gfCNCPoint2[6043] = {X 559.9503, Y 48.1273, Z -2.1667, A 0.000, B 0.000, C 0.000 }
gfCNCPoint2[6044] = {X 559.3170, Y 47.4940, Z -2.1667, A 0.000, B 0.000, C 0.000 }
gfCNCPoint2[6045] = {X 558.8404, Y 46.7355, Z -2.1667, A 0.000, B 0.000, C 0.000 }
gfCNCPoint2[6046] = {X 558.5446, Y 45.8901, Z -2.1667, A 0.000, B 0.000, C 0.000 }
gfCNCPoint2[6047] = {X 558.4443, Y 45.0000, Z -2.1667, A 0.000, B 0.000, C 0.000 }
gfCNCPoint2[6048] = {X 558.4443, Y 44.0660, Z -2.1667, A 0.000, B 0.000, C 0.000 }
gfCNCPoint2[6049] = {X 558.5395, Y 43.2139, Z -2.1667, A 0.000, B 0.000, C 0.000 }
gfCNCPoint2[6050] = {X 558.8124, Y 42.4011, Z -2.1667, A 0.000, B 0.000, C 0.000 }
gfCNCPoint2[6051] = {X 559.2508, Y 41.6643, Z -2.1667, A 0.000, B 0.000, C 0.000 }
gfCNCPoint2[6052] = {X 559.8349, Y 41.0367, Z -2.1667, A 0.000, B 0.000, C 0.000 }
gfCNCPoint2[6053] = {X 559.9032, Y 40.9788, Z -2.1667, A 0.000, B 0.000, C 0.000 }
gfCNCPoint2[6054] = {X 559.9727, Y 40.9224, Z -2.1667, A 0.000, B 0.000, C 0.000 }
gfCNCPoint2[6055] = {X 559.9727, Y 9.0791, Z -2.1667, A 0.000, B 0.000, C 0.000 }
gfCNCPoint2[6056] = {X 559.9026, Y 9.0227, Z -2.1667, A 0.000, B 0.000, C 0.000 }
gfCNCPoint2[6057] = {X 559.8337, Y 8.9647, Z -2.1667, A 0.000, B 0.000, C 0.000 }
gfCNCPoint2[6058] = {X 559.2474, Y 8.3382, Z -2.1667, A 0.000, B 0.000, C 0.000 }
gfCNCPoint2[6059] = {X 558.8082, Y 7.6010, Z -2.1667, A 0.000, B 0.000, C 0.000 }
gfCNCPoint2[6060] = {X 558.5363, Y 6.7871, Z -2.1667, A 0.000, B 0.000, C 0.000 }
gfCNCPoint2[6061] = {X 558.4443, Y 5.9339, Z -2.1667, A 0.000, B 0.000, C 0.000 }
gfCNCPoint2[6062] = {X 558.4443, Y 5.0000, Z -2.1667, A 0.000, B 0.000, C 0.000 }
gfCNCPoint2[6063] = {X 558.5446, Y 4.1099, Z -2.1667, A 0.000, B 0.000, C 0.000 }
gfCNCPoint2[6064] = {X 558.8404, Y 3.2645, Z -2.1667, A 0.000, B 0.000, C 0.000 }
gfCNCPoint2[6065] = {X 559.3170, Y 2.5060, Z -2.1667, A 0.000, B 0.000, C 0.000 }
gfCNCPoint2[6066] = {X 559.9503, Y 1.8727, Z -2.1667, A 0.000, B 0.000, C 0.000 }
gfCNCPoint2[6067] = {X 560.7088, Y 1.3961, Z -2.1667, A 0.000, B 0.000, C 0.000 }
gfCNCPoint2[6068] = {X 561.5542, Y 1.1003, Z -2.1667, A 0.000, B 0.000, C 0.000 }
gfCNCPoint2[6069] = {X 562.4443, Y 1.0000, Z -2.1667, A 0.000, B 0.000, C 0.000 }
gfCNCPoint2[6070] = {X 570.9376, Y 1.0000, Z -2.1667, A 0.000, B 0.000, C 0.000 }
gfCNCPoint2[6071] = {X 571.8276, Y 1.1003, Z -2.1667, A 0.000, B 0.000, C 0.000 }
gfCNCPoint2[6072] = {X 572.6731, Y 1.3961, Z -2.1667, A 0.000, B 0.000, C 0.000 }
gfCNCPoint2[6073] = {X 573.4315, Y 1.8727, Z -2.1667, A 0.000, B 0.000, C 0.000 }
gfCNCPoint2[6074] = {X 574.0649, Y 2.5060, Z -2.1667, A 0.000, B 0.000, C 0.000 }
gfCNCPoint2[6075] = {X 574.5414, Y 3.2645, Z -2.1667, A 0.000, B 0.000, C 0.000 }
gfCNCPoint2[6076] = {X 574.8373, Y 4.1099, Z -2.1667, A 0.000, B 0.000, C 0.000 }
gfCNCPoint2[6077] = {X 574.9376, Y 5.0000, Z -2.1667, A 0.000, B 0.000, C 0.000 }
gfCNCPoint2[6078] = {X 574.9372, Y 5.9858, Z -2.1667, A 0.000, B 0.000, C 0.000 }
gfCNCPoint2[6079] = {X 574.8649, Y 6.6932, Z -2.1667, A 0.000, B 0.000, C 0.000 }
gfCNCPoint2[6080] = {X 574.6684, Y 7.3766, Z -2.1667, A 0.000, B 0.000, C 0.000 }
gfCNCPoint2[6081] = {X 574.3540, Y 8.0145, Z -2.1667, A 0.000, B 0.000, C 0.000 }
gfCNCPoint2[6082] = {X 574.2916, Y 8.1136, Z -2.1667, A 0.000, B 0.000, C 0.000 }
gfCNCPoint2[6083] = {X 574.2264, Y 8.2108, Z -2.1667, A 0.000, B 0.000, C 0.000 }
gfCNCPoint2[6084] = {X 574.2604, Y 8.2360, Z -2.1667, A 0.000, B 0.000, C 0.000 }
gfCNCPoint2[6085] = {X 574.2832, Y 8.2715, Z -2.1667, A 0.000, B 0.000, C 0.000 }
gfCNCPoint2[6086] = {X 574.9161, Y 9.8088, Z -2.1667, A 0.000, B 0.000, C 0.000 }
gfCNCPoint2[6087] = {X 581.1904, Y 25.2176, Z -2.1667, A 0.000, B 0.000, C 0.000 }
gfCNCPoint2[6088] = {X 588.2030, Y 8.0669, Z -2.1667, A 0.000, B 0.000, C 0.000 }
gfCNCPoint2[6089] = {X 587.8648, Y 7.3988, Z -2.1667, A 0.000, B 0.000, C 0.000 }
gfCNCPoint2[6090] = {X 587.6570, Y 6.6794, Z -2.1667, A 0.000, B 0.000, C 0.000 }
gfCNCPoint2[6091] = {X 587.5870, Y 5.9339, Z -2.1667, A 0.000, B 0.000, C 0.000 }
gfCNCPoint2[6092] = {X 587.5870, Y 5.0000, Z -2.1667, A 0.000, B 0.000, C 0.000 }
gfCNCPoint2[6093] = {X 587.6872, Y 4.1099, Z -2.1667, A 0.000, B 0.000, C 0.000 }
gfCNCPoint2[6094] = {X 587.9831, Y 3.2645, Z -2.1667, A 0.000, B 0.000, C 0.000 }
gfCNCPoint2[6095] = {X 588.4596, Y 2.5060, Z -2.1667, A 0.000, B 0.000, C 0.000 }
gfCNCPoint2[6096] = {X 589.0930, Y 1.8727, Z -2.1667, A 0.000, B 0.000, C 0.000 }
gfCNCPoint2[6097] = {X 589.8514, Y 1.3961, Z -2.1667, A 0.000, B 0.000, C 0.000 }
gfCNCPoint2[6098] = {X 590.6969, Y 1.1003, Z -2.1667, A 0.000, B 0.000, C 0.000 }
gfCNCPoint2[6099] = {X 591.5870, Y 1.0000, Z -2.1667, A 0.000, B 0.000, C 0.000 }
gfCNCPoint2[6100] = {X 600.0000, Y 1.0000, Z -2.1667, A 0.000, B 0.000, C 0.000 }
gfCNCPoint2[6101] = {X 600.7927, Y 1.0793, Z -2.1667, A 0.000, B 0.000, C 0.000 }
gfCNCPoint2[6102] = {X 601.5540, Y 1.3142, Z -2.1667, A 0.000, B 0.000, C 0.000 }
gfCNCPoint2[6103] = {X 602.2536, Y 1.6953, Z -2.1667, A 0.000, B 0.000, C 0.000 }
gfCNCPoint2[6104] = {X 602.8638, Y 2.2074, Z -2.1667, A 0.000, B 0.000, C 0.000 }
gfCNCPoint2[6105] = {X 603.3604, Y 2.8303, Z -2.1667, A 0.000, B 0.000, C 0.000 }
gfCNCPoint2[6106] = {X 603.5430, Y 3.1434, Z -2.1667, A 0.000, B 0.000, C 0.000 }
gfCNCPoint2[6107] = {X 603.6965, Y 3.4716, Z -2.1667, A 0.000, B 0.000, C 0.000 }
gfCNCPoint2[6108] = {X 607.6965, Y 13.1458, Z -2.1667, A 0.000, B 0.000, C 0.000 }
gfCNCPoint2[6109] = {X 607.6965, Y 13.1458, Z 0.8333, A 0.000, B 0.000, C 0.000 }
gfCNCPoint2[6110] = {X 607.6965, Y 13.1458, Z 11.0000, A 0.000, B 0.000, C 0.000 }
gfCNCPoint2[6111] = {X 448.7118, Y 19.7811, Z 11.0000, A 0.000, B 0.000, C 0.000 }
gfCNCPoint2[6112] = {X 448.7118, Y 19.7811, Z 1.6667, A 0.000, B 0.000, C 0.000 }
gfCNCPoint2[6113] = {X 444.0413, Y 19.7808, Z 0.4152, A 0.000, B 0.000, C 0.000 }
gfCNCPoint2[6114] = {X 443.3489, Y 19.7970, Z 0.2296, A 0.000, B 0.000, C 0.000 }
gfCNCPoint2[6115] = {X 442.7481, Y 19.8041, Z 0.0686, A 0.000, B 0.000, C 0.000 }
gfCNCPoint2[6116] = {X 442.0371, Y 19.9272, Z -0.1247, A 0.000, B 0.000, C 0.000 }
gfCNCPoint2[6117] = {X 441.4689, Y 20.1225, Z -0.2857, A 0.000, B 0.000, C 0.000 }
gfCNCPoint2[6118] = {X 441.3658, Y 20.1579, Z -0.3149, A 0.000, B 0.000, C 0.000 }
gfCNCPoint2[6119] = {X 441.3328, Y 20.2618, Z -0.3441, A 0.000, B 0.000, C 0.000 }
gfCNCPoint2[6120] = {X 441.1879, Y 20.7173, Z -0.4722, A 0.000, B 0.000, C 0.000 }
gfCNCPoint2[6121] = {X 441.1541, Y 21.8891, Z -0.7863, A 0.000, B 0.000, C 0.000 }
gfCNCPoint2[6122] = {X 441.2726, Y 22.3522, Z -0.9144, A 0.000, B 0.000, C 0.000 }
gfCNCPoint2[6123] = {X 441.5010, Y 22.4270, Z -0.9788, A 0.000, B 0.000, C 0.000 }
gfCNCPoint2[6124] = {X 441.7404, Y 22.4490, Z -1.0432, A 0.000, B 0.000, C 0.000 }
gfCNCPoint2[6125] = {X 442.9814, Y 22.5631, Z -1.3771, A 0.000, B 0.000, C 0.000 }
gfCNCPoint2[6126] = {X 443.1437, Y 22.5696, Z -1.4207, A 0.000, B 0.000, C 0.000 }
gfCNCPoint2[6127] = {X 444.3942, Y 22.5560, Z -1.7558, A 0.000, B 0.000, C 0.000 }
gfCNCPoint2[6128] = {X 445.9278, Y 22.5560, Z -2.1667, A 0.000, B 0.000, C 0.000 }
gfCNCPoint2[6129] = {X 450.1184, Y 22.5560, Z -2.1667, A 0.000, B 0.000, C 0.000 }
gfCNCPoint2[6130] = {X 450.1184, Y 19.7812, Z -2.1667, A 0.000, B 0.000, C 0.000 }
gfCNCPoint2[6131] = {X 444.0413, Y 19.7808, Z -2.1667, A 0.000, B 0.000, C 0.000 }
gfCNCPoint2[6132] = {X 443.3489, Y 19.7970, Z -2.1667, A 0.000, B 0.000, C 0.000 }
gfCNCPoint2[6133] = {X 442.3959, Y 19.8846, Z -2.1667, A 0.000, B 0.000, C 0.000 }
gfCNCPoint2[6134] = {X 441.4689, Y 20.1225, Z -2.1667, A 0.000, B 0.000, C 0.000 }
gfCNCPoint2[6135] = {X 441.3843, Y 20.1760, Z -2.1667, A 0.000, B 0.000, C 0.000 }
gfCNCPoint2[6136] = {X 441.3328, Y 20.2618, Z -2.1667, A 0.000, B 0.000, C 0.000 }
gfCNCPoint2[6137] = {X 441.1824, Y 20.9508, Z -2.1667, A 0.000, B 0.000, C 0.000 }
gfCNCPoint2[6138] = {X 441.1621, Y 21.6557, Z -2.1667, A 0.000, B 0.000, C 0.000 }
gfCNCPoint2[6139] = {X 441.2726, Y 22.3522, Z -2.1667, A 0.000, B 0.000, C 0.000 }
gfCNCPoint2[6140] = {X 441.5038, Y 22.4137, Z -2.1667, A 0.000, B 0.000, C 0.000 }
gfCNCPoint2[6141] = {X 441.7404, Y 22.4490, Z -2.1667, A 0.000, B 0.000, C 0.000 }
gfCNCPoint2[6142] = {X 443.0660, Y 22.5366, Z -2.1667, A 0.000, B 0.000, C 0.000 }
gfCNCPoint2[6143] = {X 444.3942, Y 22.5560, Z -2.1667, A 0.000, B 0.000, C 0.000 }
gfCNCPoint2[6144] = {X 445.9278, Y 22.5560, Z -2.1667, A 0.000, B 0.000, C 0.000 }
gfCNCPoint2[6145] = {X 441.9430, Y 22.2874, Z -2.1667, A 0.000, B 0.000, C 0.000 }
gfCNCPoint2[6146] = {X 445.9278, Y 22.6360, Z -2.1667, A 0.000, B 0.000, C 0.000 }
gfCNCPoint2[6147] = {X 450.1984, Y 22.6360, Z -2.1667, A 0.000, B 0.000, C 0.000 }
gfCNCPoint2[6148] = {X 450.1984, Y 19.7012, Z -2.1667, A 0.000, B 0.000, C 0.000 }
gfCNCPoint2[6149] = {X 444.0404, Y 19.7008, Z -2.1667, A 0.000, B 0.000, C 0.000 }
gfCNCPoint2[6150] = {X 443.3498, Y 19.7169, Z -2.1667, A 0.000, B 0.000, C 0.000 }
gfCNCPoint2[6151] = {X 442.3831, Y 19.8056, Z -2.1667, A 0.000, B 0.000, C 0.000 }
gfCNCPoint2[6152] = {X 441.4429, Y 20.0469, Z -2.1667, A 0.000, B 0.000, C 0.000 }
gfCNCPoint2[6153] = {X 441.3271, Y 20.1201, Z -2.1667, A 0.000, B 0.000, C 0.000 }
gfCNCPoint2[6154] = {X 441.2566, Y 20.2375, Z -2.1667, A 0.000, B 0.000, C 0.000 }
gfCNCPoint2[6155] = {X 441.1012, Y 20.9555, Z -2.1667, A 0.000, B 0.000, C 0.000 }
gfCNCPoint2[6156] = {X 441.0842, Y 21.6898, Z -2.1667, A 0.000, B 0.000, C 0.000 }
gfCNCPoint2[6157] = {X 441.2061, Y 22.4142, Z -2.1667, A 0.000, B 0.000, C 0.000 }
gfCNCPoint2[6158] = {X 441.4661, Y 22.4875, Z -2.1667, A 0.000, B 0.000, C 0.000 }
gfCNCPoint2[6159] = {X 441.7331, Y 22.5286, Z -2.1667, A 0.000, B 0.000, C 0.000 }
gfCNCPoint2[6160] = {X 443.0614, Y 22.6165, Z -2.1667, A 0.000, B 0.000, C 0.000 }
gfCNCPoint2[6161] = {X 444.3925, Y 22.6360, Z -2.1667, A 0.000, B 0.000, C 0.000 }
gfCNCPoint2[6162] = {X 445.9278, Y 22.6360, Z -2.1667, A 0.000, B 0.000, C 0.000 }
gfCNCPoint2[6163] = {X 449.9125, Y 22.2874, Z -2.1667, A 0.000, B 0.000, C 0.000 }
gfCNCPoint2[6164] = {X 441.9430, Y 22.3674, Z -2.1667, A 0.000, B 0.000, C 0.000 }
gfCNCPoint2[6165] = {X 445.9278, Y 22.7160, Z -2.1667, A 0.000, B 0.000, C 0.000 }
gfCNCPoint2[6166] = {X 450.2784, Y 22.7160, Z -2.1667, A 0.000, B 0.000, C 0.000 }
gfCNCPoint2[6167] = {X 450.2784, Y 19.6212, Z -2.1667, A 0.000, B 0.000, C 0.000 }
gfCNCPoint2[6168] = {X 444.0395, Y 19.6208, Z -2.1667, A 0.000, B 0.000, C 0.000 }
gfCNCPoint2[6169] = {X 443.3484, Y 19.6370, Z -2.1667, A 0.000, B 0.000, C 0.000 }
gfCNCPoint2[6170] = {X 442.3693, Y 19.7268, Z -2.1667, A 0.000, B 0.000, C 0.000 }
gfCNCPoint2[6171] = {X 441.4169, Y 19.9712, Z -2.1667, A 0.000, B 0.000, C 0.000 }
gfCNCPoint2[6172] = {X 441.2699, Y 20.0642, Z -2.1667, A 0.000, B 0.000, C 0.000 }
gfCNCPoint2[6173] = {X 441.1803, Y 20.2133, Z -2.1667, A 0.000, B 0.000, C 0.000 }
gfCNCPoint2[6174] = {X 441.0202, Y 20.9599, Z -2.1667, A 0.000, B 0.000, C 0.000 }
gfCNCPoint2[6175] = {X 441.0065, Y 21.7235, Z -2.1667, A 0.000, B 0.000, C 0.000 }
gfCNCPoint2[6176] = {X 441.1399, Y 22.4754, Z -2.1667, A 0.000, B 0.000, C 0.000 }
gfCNCPoint2[6177] = {X 441.4285, Y 22.5611, Z -2.1667, A 0.000, B 0.000, C 0.000 }
gfCNCPoint2[6178] = {X 441.7258, Y 22.6083, Z -2.1667, A 0.000, B 0.000, C 0.000 }
gfCNCPoint2[6179] = {X 443.0580, Y 22.6964, Z -2.1667, A 0.000, B 0.000, C 0.000 }
gfCNCPoint2[6180] = {X 444.3929, Y 22.7160, Z -2.1667, A 0.000, B 0.000, C 0.000 }
gfCNCPoint2[6181] = {X 445.9278, Y 22.7160, Z -2.1667, A 0.000, B 0.000, C 0.000 }
gfCNCPoint2[6182] = {X 449.9125, Y 22.3674, Z -2.1667, A 0.000, B 0.000, C 0.000 }
gfCNCPoint2[6183] = {X 441.9430, Y 22.4474, Z -2.1667, A 0.000, B 0.000, C 0.000 }
gfCNCPoint2[6184] = {X 445.9278, Y 22.7960, Z -2.1667, A 0.000, B 0.000, C 0.000 }
gfCNCPoint2[6185] = {X 450.3584, Y 22.7960, Z -2.1667, A 0.000, B 0.000, C 0.000 }
gfCNCPoint2[6186] = {X 450.3584, Y 19.5412, Z -2.1667, A 0.000, B 0.000, C 0.000 }
gfCNCPoint2[6187] = {X 444.0385, Y 19.5408, Z -2.1667, A 0.000, B 0.000, C 0.000 }
gfCNCPoint2[6188] = {X 443.3470, Y 19.5570, Z -2.1667, A 0.000, B 0.000, C 0.000 }
gfCNCPoint2[6189] = {X 442.3554, Y 19.6480, Z -2.1667, A 0.000, B 0.000, C 0.000 }
gfCNCPoint2[6190] = {X 441.3909, Y 19.8955, Z -2.1667, A 0.000, B 0.000, C 0.000 }
gfCNCPoint2[6191] = {X 441.2127, Y 20.0083, Z -2.1667, A 0.000, B 0.000, C 0.000 }
gfCNCPoint2[6192] = {X 441.1041, Y 20.1890, Z -2.1667, A 0.000, B 0.000, C 0.000 }
gfCNCPoint2[6193] = {X 440.9392, Y 20.9642, Z -2.1667, A 0.000, B 0.000, C 0.000 }
gfCNCPoint2[6194] = {X 440.9290, Y 21.7567, Z -2.1667, A 0.000, B 0.000, C 0.000 }
gfCNCPoint2[6195] = {X 441.0740, Y 22.5359, Z -2.1667, A 0.000, B 0.000, C 0.000 }
gfCNCPoint2[6196] = {X 441.3909, Y 22.6345, Z -2.1667, A 0.000, B 0.000, C 0.000 }
gfCNCPoint2[6197] = {X 441.7184, Y 22.6880, Z -2.1667, A 0.000, B 0.000, C 0.000 }
gfCNCPoint2[6198] = {X 443.0545, Y 22.7763, Z -2.1667, A 0.000, B 0.000, C 0.000 }
gfCNCPoint2[6199] = {X 444.3934, Y 22.7960, Z -2.1667, A 0.000, B 0.000, C 0.000 }
gfCNCPoint2[6200] = {X 445.9278, Y 22.7960, Z -2.1667, A 0.000, B 0.000, C 0.000 }
gfCNCPoint2[6201] = {X 449.9125, Y 22.4474, Z -2.1667, A 0.000, B 0.000, C 0.000 }
gfCNCPoint2[6202] = {X 441.9430, Y 22.5274, Z -2.1667, A 0.000, B 0.000, C 0.000 }
gfCNCPoint2[6203] = {X 445.9278, Y 22.8760, Z -2.1667, A 0.000, B 0.000, C 0.000 }
gfCNCPoint2[6204] = {X 450.4384, Y 22.8760, Z -2.1667, A 0.000, B 0.000, C 0.000 }
gfCNCPoint2[6205] = {X 450.4384, Y 19.4612, Z -2.1667, A 0.000, B 0.000, C 0.000 }
gfCNCPoint2[6206] = {X 444.0376, Y 19.4608, Z -2.1667, A 0.000, B 0.000, C 0.000 }
gfCNCPoint2[6207] = {X 443.3456, Y 19.4770, Z -2.1667, A 0.000, B 0.000, C 0.000 }
gfCNCPoint2[6208] = {X 442.3415, Y 19.5692, Z -2.1667, A 0.000, B 0.000, C 0.000 }
gfCNCPoint2[6209] = {X 441.3649, Y 19.8199, Z -2.1667, A 0.000, B 0.000, C 0.000 }
gfCNCPoint2[6210] = {X 441.1555, Y 19.9524, Z -2.1667, A 0.000, B 0.000, C 0.000 }
gfCNCPoint2[6211] = {X 441.0279, Y 20.1648, Z -2.1667, A 0.000, B 0.000, C 0.000 }
gfCNCPoint2[6212] = {X 440.8582, Y 20.9683, Z -2.1667, A 0.000, B 0.000, C 0.000 }
gfCNCPoint2[6213] = {X 440.8516, Y 21.7896, Z -2.1667, A 0.000, B 0.000, C 0.000 }
gfCNCPoint2[6214] = {X 441.0082, Y 22.5958, Z -2.1667, A 0.000, B 0.000, C 0.000 }
gfCNCPoint2[6215] = {X 441.3533, Y 22.7078, Z -2.1667, A 0.000, B 0.000, C 0.000 }
gfCNCPoint2[6216] = {X 441.7111, Y 22.7676, Z -2.1667, A 0.000, B 0.000, C 0.000 }
gfCNCPoint2[6217] = {X 443.0511, Y 22.8562, Z -2.1667, A 0.000, B 0.000, C 0.000 }
gfCNCPoint2[6218] = {X 444.3938, Y 22.8760, Z -2.1667, A 0.000, B 0.000, C 0.000 }
gfCNCPoint2[6219] = {X 445.9278, Y 22.8760, Z -2.1667, A 0.000, B 0.000, C 0.000 }
gfCNCPoint2[6220] = {X 449.9125, Y 22.5274, Z -2.1667, A 0.000, B 0.000, C 0.000 }
gfCNCPoint2[6221] = {X 441.9430, Y 22.6074, Z -2.1667, A 0.000, B 0.000, C 0.000 }
gfCNCPoint2[6222] = {X 445.9278, Y 22.9560, Z -2.1667, A 0.000, B 0.000, C 0.000 }
gfCNCPoint2[6223] = {X 450.5184, Y 22.9560, Z -2.1667, A 0.000, B 0.000, C 0.000 }
gfCNCPoint2[6224] = {X 450.5197, Y 19.3812, Z -2.1667, A 0.000, B 0.000, C 0.000 }
gfCNCPoint2[6225] = {X 444.0367, Y 19.3808, Z -2.1667, A 0.000, B 0.000, C 0.000 }
gfCNCPoint2[6226] = {X 443.3442, Y 19.3970, Z -2.1667, A 0.000, B 0.000, C 0.000 }
gfCNCPoint2[6227] = {X 442.3276, Y 19.4904, Z -2.1667, A 0.000, B 0.000, C 0.000 }
gfCNCPoint2[6228] = {X 441.3389, Y 19.7442, Z -2.1667, A 0.000, B 0.000, C 0.000 }
gfCNCPoint2[6229] = {X 441.0982, Y 19.8964, Z -2.1667, A 0.000, B 0.000, C 0.000 }
gfCNCPoint2[6230] = {X 440.9516, Y 20.1405, Z -2.1667, A 0.000, B 0.000, C 0.000 }
gfCNCPoint2[6231] = {X 440.7773, Y 20.9723, Z -2.1667, A 0.000, B 0.000, C 0.000 }
gfCNCPoint2[6232] = {X 440.7743, Y 21.8221, Z -2.1667, A 0.000, B 0.000, C 0.000 }
gfCNCPoint2[6233] = {X 440.9427, Y 22.6551, Z -2.1667, A 0.000, B 0.000, C 0.000 }
gfCNCPoint2[6234] = {X 441.3158, Y 22.7809, Z -2.1667, A 0.000, B 0.000, C 0.000 }
gfCNCPoint2[6235] = {X 441.7038, Y 22.8473, Z -2.1667, A 0.000, B 0.000, C 0.000 }
gfCNCPoint2[6236] = {X 443.0476, Y 22.9362, Z -2.1667, A 0.000, B 0.000, C 0.000 }
gfCNCPoint2[6237] = {X 444.3942, Y 22.9560, Z -2.1667, A 0.000, B 0.000, C 0.000 }
gfCNCPoint2[6238] = {X 445.9278, Y 22.9560, Z -2.1667, A 0.000, B 0.000, C 0.000 }
gfCNCPoint2[6239] = {X 449.9125, Y 22.6074, Z -2.1667, A 0.000, B 0.000, C 0.000 }
gfCNCPoint2[6240] = {X 449.9125, Y 22.6074, Z 0.8333, A 0.000, B 0.000, C 0.000 }
gfCNCPoint2[6241] = {X 449.9125, Y 22.6074, Z 11.0000, A 0.000, B 0.000, C 0.000 }
gfCNCPoint2[6242] = {X 492.1935, Y 19.7809, Z 11.0000, A 0.000, B 0.000, C 0.000 }
gfCNCPoint2[6243] = {X 492.1935, Y 19.7809, Z 1.6667, A 0.000, B 0.000, C 0.000 }
gfCNCPoint2[6244] = {X 487.6645, Y 19.7801, Z 0.4531, A 0.000, B 0.000, C 0.000 }
gfCNCPoint2[6245] = {X 486.9699, Y 19.7848, Z 0.2670, A 0.000, B 0.000, C 0.000 }
gfCNCPoint2[6246] = {X 486.2675, Y 19.7834, Z 0.0788, A 0.000, B 0.000, C 0.000 }
gfCNCPoint2[6247] = {X 485.4755, Y 19.8884, Z -0.1353, A 0.000, B 0.000, C 0.000 }
gfCNCPoint2[6248] = {X 484.7978, Y 20.0729, Z -0.3235, A 0.000, B 0.000, C 0.000 }
gfCNCPoint2[6249] = {X 484.6638, Y 20.1094, Z -0.3607, A 0.000, B 0.000, C 0.000 }
gfCNCPoint2[6250] = {X 484.6332, Y 20.1381, Z -0.3719, A 0.000, B 0.000, C 0.000 }
gfCNCPoint2[6251] = {X 484.5883, Y 20.2695, Z -0.4091, A 0.000, B 0.000, C 0.000 }
gfCNCPoint2[6252] = {X 484.4391, Y 20.7065, Z -0.5329, A 0.000, B 0.000, C 0.000 }
gfCNCPoint2[6253] = {X 484.4034, Y 21.9102, Z -0.8555, A 0.000, B 0.000, C 0.000 }
gfCNCPoint2[6254] = {X 484.5263, Y 22.3553, Z -0.9793, A 0.000, B 0.000, C 0.000 }
gfCNCPoint2[6255] = {X 484.6983, Y 22.4113, Z -1.0277, A 0.000, B 0.000, C 0.000 }
gfCNCPoint2[6256] = {X 484.8781, Y 22.4311, Z -1.0762, A 0.000, B 0.000, C 0.000 }
gfCNCPoint2[6257] = {X 486.0368, Y 22.5560, Z -1.3885, A 0.000, B 0.000, C 0.000 }
gfCNCPoint2[6258] = {X 487.1542, Y 22.5560, Z -1.6879, A 0.000, B 0.000, C 0.000 }
gfCNCPoint2[6259] = {X 488.9410, Y 22.5560, Z -2.1667, A 0.000, B 0.000, C 0.000 }
gfCNCPoint2[6260] = {X 493.3690, Y 22.5560, Z -2.1667, A 0.000, B 0.000, C 0.000 }
gfCNCPoint2[6261] = {X 493.3690, Y 19.7811, Z -2.1667, A 0.000, B 0.000, C 0.000 }
gfCNCPoint2[6262] = {X 487.6645, Y 19.7801, Z -2.1667, A 0.000, B 0.000, C 0.000 }
gfCNCPoint2[6263] = {X 486.9699, Y 19.7848, Z -2.1667, A 0.000, B 0.000, C 0.000 }
gfCNCPoint2[6264] = {X 485.8742, Y 19.8560, Z -2.1667, A 0.000, B 0.000, C 0.000 }
gfCNCPoint2[6265] = {X 484.7978, Y 20.0729, Z -2.1667, A 0.000, B 0.000, C 0.000 }
gfCNCPoint2[6266] = {X 484.6686, Y 20.1452, Z -2.1667, A 0.000, B 0.000, C 0.000 }
gfCNCPoint2[6267] = {X 484.5883, Y 20.2695, Z -2.1667, A 0.000, B 0.000, C 0.000 }
gfCNCPoint2[6268] = {X 484.4281, Y 20.9560, Z -2.1667, A 0.000, B 0.000, C 0.000 }
gfCNCPoint2[6269] = {X 484.4072, Y 21.6606, Z -2.1667, A 0.000, B 0.000, C 0.000 }
gfCNCPoint2[6270] = {X 484.5263, Y 22.3553, Z -2.1667, A 0.000, B 0.000, C 0.000 }
gfCNCPoint2[6271] = {X 484.7003, Y 22.4022, Z -2.1667, A 0.000, B 0.000, C 0.000 }
gfCNCPoint2[6272] = {X 484.8781, Y 22.4311, Z -2.1667, A 0.000, B 0.000, C 0.000 }
gfCNCPoint2[6273] = {X 486.0144, Y 22.5248, Z -2.1667, A 0.000, B 0.000, C 0.000 }
gfCNCPoint2[6274] = {X 487.1542, Y 22.5560, Z -2.1667, A 0.000, B 0.000, C 0.000 }
gfCNCPoint2[6275] = {X 488.9410, Y 22.5560, Z -2.1667, A 0.000, B 0.000, C 0.000 }
gfCNCPoint2[6276] = {X 484.9563, Y 22.2874, Z -2.1667, A 0.000, B 0.000, C 0.000 }
gfCNCPoint2[6277] = {X 488.9410, Y 22.6360, Z -2.1667, A 0.000, B 0.000, C 0.000 }
gfCNCPoint2[6278] = {X 493.4490, Y 22.6360, Z -2.1667, A 0.000, B 0.000, C 0.000 }
gfCNCPoint2[6279] = {X 493.4490, Y 19.7011, Z -2.1667, A 0.000, B 0.000, C 0.000 }
gfCNCPoint2[6280] = {X 487.6642, Y 19.7001, Z -2.1667, A 0.000, B 0.000, C 0.000 }
gfCNCPoint2[6281] = {X 486.9714, Y 19.7048, Z -2.1667, A 0.000, B 0.000, C 0.000 }
gfCNCPoint2[6282] = {X 485.8643, Y 19.7767, Z -2.1667, A 0.000, B 0.000, C 0.000 }
gfCNCPoint2[6283] = {X 484.7768, Y 19.9957, Z -2.1667, A 0.000, B 0.000, C 0.000 }
gfCNCPoint2[6284] = {X 484.6138, Y 20.0868, Z -2.1667, A 0.000, B 0.000, C 0.000 }
gfCNCPoint2[6285] = {X 484.5126, Y 20.2437, Z -2.1667, A 0.000, B 0.000, C 0.000 }
gfCNCPoint2[6286] = {X 484.3470, Y 20.9597, Z -2.1667, A 0.000, B 0.000, C 0.000 }
gfCNCPoint2[6287] = {X 484.3295, Y 21.6945, Z -2.1667, A 0.000, B 0.000, C 0.000 }
gfCNCPoint2[6288] = {X 484.4608, Y 22.4176, Z -2.1667, A 0.000, B 0.000, C 0.000 }
gfCNCPoint2[6289] = {X 484.6624, Y 22.4758, Z -2.1667, A 0.000, B 0.000, C 0.000 }
gfCNCPoint2[6290] = {X 484.8693, Y 22.5106, Z -2.1667, A 0.000, B 0.000, C 0.000 }
gfCNCPoint2[6291] = {X 486.0100, Y 22.6047, Z -2.1667, A 0.000, B 0.000, C 0.000 }
gfCNCPoint2[6292] = {X 487.1542, Y 22.6360, Z -2.1667, A 0.000, B 0.000, C 0.000 }
gfCNCPoint2[6293] = {X 488.9410, Y 22.6360, Z -2.1667, A 0.000, B 0.000, C 0.000 }
gfCNCPoint2[6294] = {X 492.9258, Y 22.2874, Z -2.1667, A 0.000, B 0.000, C 0.000 }
gfCNCPoint2[6295] = {X 484.9563, Y 22.3674, Z -2.1667, A 0.000, B 0.000, C 0.000 }
gfCNCPoint2[6296] = {X 488.9410, Y 22.7160, Z -2.1667, A 0.000, B 0.000, C 0.000 }
gfCNCPoint2[6297] = {X 493.5290, Y 22.7160, Z -2.1667, A 0.000, B 0.000, C 0.000 }
gfCNCPoint2[6298] = {X 493.5290, Y 19.6212, Z -2.1667, A 0.000, B 0.000, C 0.000 }
gfCNCPoint2[6299] = {X 487.6640, Y 19.6201, Z -2.1667, A 0.000, B 0.000, C 0.000 }
gfCNCPoint2[6300] = {X 486.9712, Y 19.6248, Z -2.1667, A 0.000, B 0.000, C 0.000 }
gfCNCPoint2[6301] = {X 485.8536, Y 19.6974, Z -2.1667, A 0.000, B 0.000, C 0.000 }
gfCNCPoint2[6302] = {X 484.7558, Y 19.9185, Z -2.1667, A 0.000, B 0.000, C 0.000 }
gfCNCPoint2[6303] = {X 484.5591, Y 20.0285, Z -2.1667, A 0.000, B 0.000, C 0.000 }
gfCNCPoint2[6304] = {X 484.4369, Y 20.2178, Z -2.1667, A 0.000, B 0.000, C 0.000 }
gfCNCPoint2[6305] = {X 484.2659, Y 20.9632, Z -2.1667, A 0.000, B 0.000, C 0.000 }
gfCNCPoint2[6306] = {X 484.2520, Y 21.7278, Z -2.1667, A 0.000, B 0.000, C 0.000 }
gfCNCPoint2[6307] = {X 484.3955, Y 22.4789, Z -2.1667, A 0.000, B 0.000, C 0.000 }
gfCNCPoint2[6308] = {X 484.6246, Y 22.5491, Z -2.1667, A 0.000, B 0.000, C 0.000 }
gfCNCPoint2[6309] = {X 484.8606, Y 22.5901, Z -2.1667, A 0.000, B 0.000, C 0.000 }
gfCNCPoint2[6310] = {X 486.0057, Y 22.6845, Z -2.1667, A 0.000, B 0.000, C 0.000 }
gfCNCPoint2[6311] = {X 487.1542, Y 22.7160, Z -2.1667, A 0.000, B 0.000, C 0.000 }
gfCNCPoint2[6312] = {X 488.9410, Y 22.7160, Z -2.1667, A 0.000, B 0.000, C 0.000 }
gfCNCPoint2[6313] = {X 492.9258, Y 22.3674, Z -2.1667, A 0.000, B 0.000, C 0.000 }
gfCNCPoint2[6314] = {X 484.9563, Y 22.4474, Z -2.1667, A 0.000, B 0.000, C 0.000 }
gfCNCPoint2[6315] = {X 488.9410, Y 22.7960, Z -2.1667, A 0.000, B 0.000, C 0.000 }
gfCNCPoint2[6316] = {X 493.6090, Y 22.7960, Z -2.1667, A 0.000, B 0.000, C 0.000 }
gfCNCPoint2[6317] = {X 493.6090, Y 19.5412, Z -2.1667, A 0.000, B 0.000, C 0.000 }
gfCNCPoint2[6318] = {X 487.6637, Y 19.5401, Z -2.1667, A 0.000, B 0.000, C 0.000 }
gfCNCPoint2[6319] = {X 486.9711, Y 19.5448, Z -2.1667, A 0.000, B 0.000, C 0.000 }
gfCNCPoint2[6320] = {X 485.8430, Y 19.6181, Z -2.1667, A 0.000, B 0.000, C 0.000 }
gfCNCPoint2[6321] = {X 484.7347, Y 19.8413, Z -2.1667, A 0.000, B 0.000, C 0.000 }
gfCNCPoint2[6322] = {X 484.5043, Y 19.9702, Z -2.1667, A 0.000, B 0.000, C 0.000 }
gfCNCPoint2[6323] = {X 484.3612, Y 20.1920, Z -2.1667, A 0.000, B 0.000, C 0.000 }
gfCNCPoint2[6324] = {X 484.1850, Y 20.9665, Z -2.1667, A 0.000, B 0.000, C 0.000 }
gfCNCPoint2[6325] = {X 484.1746, Y 21.7607, Z -2.1667, A 0.000, B 0.000, C 0.000 }
gfCNCPoint2[6326] = {X 484.3304, Y 22.5395, Z -2.1667, A 0.000, B 0.000, C 0.000 }
gfCNCPoint2[6327] = {X 484.5867, Y 22.6222, Z -2.1667, A 0.000, B 0.000, C 0.000 }
gfCNCPoint2[6328] = {X 484.8518, Y 22.6697, Z -2.1667, A 0.000, B 0.000, C 0.000 }
gfCNCPoint2[6329] = {X 486.0013, Y 22.7644, Z -2.1667, A 0.000, B 0.000, C 0.000 }
gfCNCPoint2[6330] = {X 487.1542, Y 22.7960, Z -2.1667, A 0.000, B 0.000, C 0.000 }
gfCNCPoint2[6331] = {X 488.9410, Y 22.7960, Z -2.1667, A 0.000, B 0.000, C 0.000 }
gfCNCPoint2[6332] = {X 492.9258, Y 22.4474, Z -2.1667, A 0.000, B 0.000, C 0.000 }
gfCNCPoint2[6333] = {X 484.9563, Y 22.5274, Z -2.1667, A 0.000, B 0.000, C 0.000 }
gfCNCPoint2[6334] = {X 488.9410, Y 22.8760, Z -2.1667, A 0.000, B 0.000, C 0.000 }
gfCNCPoint2[6335] = {X 493.6890, Y 22.8760, Z -2.1667, A 0.000, B 0.000, C 0.000 }
gfCNCPoint2[6336] = {X 493.6890, Y 19.4612, Z -2.1667, A 0.000, B 0.000, C 0.000 }
gfCNCPoint2[6337] = {X 487.6634, Y 19.4601, Z -2.1667, A 0.000, B 0.000, C 0.000 }
gfCNCPoint2[6338] = {X 486.9709, Y 19.4648, Z -2.1667, A 0.000, B 0.000, C 0.000 }
gfCNCPoint2[6339] = {X 485.8323, Y 19.5388, Z -2.1667, A 0.000, B 0.000, C 0.000 }
gfCNCPoint2[6340] = {X 484.7137, Y 19.7642, Z -2.1667, A 0.000, B 0.000, C 0.000 }
gfCNCPoint2[6341] = {X 484.4496, Y 19.9118, Z -2.1667, A 0.000, B 0.000, C 0.000 }
gfCNCPoint2[6342] = {X 484.2855, Y 20.1662, Z -2.1667, A 0.000, B 0.000, C 0.000 }
gfCNCPoint2[6343] = {X 484.1041, Y 20.9695, Z -2.1667, A 0.000, B 0.000, C 0.000 }
gfCNCPoint2[6344] = {X 484.0973, Y 21.7931, Z -2.1667, A 0.000, B 0.000, C 0.000 }
gfCNCPoint2[6345] = {X 484.2655, Y 22.5994, Z -2.1667, A 0.000, B 0.000, C 0.000 }
gfCNCPoint2[6346] = {X 484.5489, Y 22.6951, Z -2.1667, A 0.000, B 0.000, C 0.000 }
gfCNCPoint2[6347] = {X 484.8431, Y 22.7492, Z -2.1667, A 0.000, B 0.000, C 0.000 }
gfCNCPoint2[6348] = {X 485.9969, Y 22.8443, Z -2.1667, A 0.000, B 0.000, C 0.000 }
gfCNCPoint2[6349] = {X 487.1542, Y 22.8760, Z -2.1667, A 0.000, B 0.000, C 0.000 }
gfCNCPoint2[6350] = {X 488.9410, Y 22.8760, Z -2.1667, A 0.000, B 0.000, C 0.000 }
gfCNCPoint2[6351] = {X 492.9258, Y 22.5274, Z -2.1667, A 0.000, B 0.000, C 0.000 }
gfCNCPoint2[6352] = {X 484.9563, Y 22.6074, Z -2.1667, A 0.000, B 0.000, C 0.000 }
gfCNCPoint2[6353] = {X 488.9410, Y 22.9560, Z -2.1667, A 0.000, B 0.000, C 0.000 }
gfCNCPoint2[6354] = {X 493.7690, Y 22.9560, Z -2.1667, A 0.000, B 0.000, C 0.000 }
gfCNCPoint2[6355] = {X 493.7702, Y 19.3812, Z -2.1667, A 0.000, B 0.000, C 0.000 }
gfCNCPoint2[6356] = {X 487.6632, Y 19.3801, Z -2.1667, A 0.000, B 0.000, C 0.000 }
gfCNCPoint2[6357] = {X 486.9707, Y 19.3848, Z -2.1667, A 0.000, B 0.000, C 0.000 }
gfCNCPoint2[6358] = {X 485.8216, Y 19.4595, Z -2.1667, A 0.000, B 0.000, C 0.000 }
gfCNCPoint2[6359] = {X 484.6927, Y 19.6870, Z -2.1667, A 0.000, B 0.000, C 0.000 }
gfCNCPoint2[6360] = {X 484.3948, Y 19.8535, Z -2.1667, A 0.000, B 0.000, C 0.000 }
gfCNCPoint2[6361] = {X 484.2098, Y 20.1403, Z -2.1667, A 0.000, B 0.000, C 0.000 }
gfCNCPoint2[6362] = {X 484.0232, Y 20.9724, Z -2.1667, A 0.000, B 0.000, C 0.000 }
gfCNCPoint2[6363] = {X 484.0202, Y 21.8252, Z -2.1667, A 0.000, B 0.000, C 0.000 }
gfCNCPoint2[6364] = {X 484.2007, Y 22.6586, Z -2.1667, A 0.000, B 0.000, C 0.000 }
gfCNCPoint2[6365] = {X 484.5110, Y 22.7679, Z -2.1667, A 0.000, B 0.000, C 0.000 }
gfCNCPoint2[6366] = {X 484.8343, Y 22.8287, Z -2.1667, A 0.000, B 0.000, C 0.000 }
gfCNCPoint2[6367] = {X 485.9925, Y 22.9242, Z -2.1667, A 0.000, B 0.000, C 0.000 }
gfCNCPoint2[6368] = {X 487.1542, Y 22.9560, Z -2.1667, A 0.000, B 0.000, C 0.000 }
gfCNCPoint2[6369] = {X 488.9410, Y 22.9560, Z -2.1667, A 0.000, B 0.000, C 0.000 }
gfCNCPoint2[6370] = {X 492.9258, Y 22.6074, Z -2.1667, A 0.000, B 0.000, C 0.000 }
gfCNCPoint2[6371] = {X 492.9258, Y 22.6074, Z 0.8333, A 0.000, B 0.000, C 0.000 }
gfCNCPoint2[6372] = {X 492.9258, Y 22.6074, Z 11.0000, A 0.000, B 0.000, C 0.000 }
gfCNCPoint2[6373] = {X 607.6965, Y 2.1254, Z 11.0000, A 0.000, B 0.000, C 0.000 }
gfCNCPoint2[6374] = {X 607.6965, Y 2.1254, Z 0.8333, A 0.000, B 0.000, C 0.000 }
gfCNCPoint2[6375] = {X 607.6965, Y 2.1254, Z -2.1667, A 0.000, B 0.000, C 0.000 }
gfCNCPoint2[6376] = {X 603.6965, Y 8.3207, Z -2.1667, A 0.000, B 0.000, C 0.000 }
gfCNCPoint2[6377] = {X 603.3201, Y 8.8215, Z -2.1667, A 0.000, B 0.000, C 0.000 }
gfCNCPoint2[6378] = {X 602.8764, Y 9.2637, Z -2.1667, A 0.000, B 0.000, C 0.000 }
gfCNCPoint2[6379] = {X 602.8763, Y 40.7363, Z -2.1667, A 0.000, B 0.000, C 0.000 }
gfCNCPoint2[6380] = {X 603.3201, Y 41.1785, Z -2.1667, A 0.000, B 0.000, C 0.000 }
gfCNCPoint2[6381] = {X 603.6965, Y 41.6793, Z -2.1667, A 0.000, B 0.000, C 0.000 }
gfCNCPoint2[6382] = {X 607.6965, Y 47.8746, Z -2.1667, A 0.000, B 0.000, C 0.000 }
gfCNCPoint2[6383] = {X 607.6965, Y 47.8746, Z 0.8333, A 0.000, B 0.000, C 0.000 }
gfCNCPoint2[6384] = {X 607.6965, Y 47.8746, Z 11.0000, A 0.000, B 0.000, C 0.000 }
gfCNCPoint2[6385] = {X 607.6965, Y 1.5516, Z 11.0000, A 0.000, B 0.000, C 0.000 }
gfCNCPoint2[6386] = {X 607.6965, Y 1.5516, Z 0.8333, A 0.000, B 0.000, C 0.000 }
gfCNCPoint2[6387] = {X 607.6965, Y 1.5516, Z -2.1667, A 0.000, B 0.000, C 0.000 }
gfCNCPoint2[6388] = {X 603.6965, Y 8.1704, Z -2.1667, A 0.000, B 0.000, C 0.000 }
gfCNCPoint2[6389] = {X 603.2892, Y 8.7356, Z -2.1667, A 0.000, B 0.000, C 0.000 }
gfCNCPoint2[6390] = {X 602.7964, Y 9.2281, Z -2.1667, A 0.000, B 0.000, C 0.000 }
gfCNCPoint2[6391] = {X 602.7963, Y 40.7726, Z -2.1667, A 0.000, B 0.000, C 0.000 }
gfCNCPoint2[6392] = {X 603.2892, Y 41.2649, Z -2.1667, A 0.000, B 0.000, C 0.000 }
gfCNCPoint2[6393] = {X 603.6965, Y 41.8300, Z -2.1667, A 0.000, B 0.000, C 0.000 }
gfCNCPoint2[6394] = {X 607.6965, Y 48.4457, Z -2.1667, A 0.000, B 0.000, C 0.000 }
gfCNCPoint2[6395] = {X 607.6965, Y 48.4457, Z 0.8333, A 0.000, B 0.000, C 0.000 }
gfCNCPoint2[6396] = {X 607.6965, Y 48.4457, Z 11.0000, A 0.000, B 0.000, C 0.000 }
gfCNCPoint2[6397] = {X 607.6965, Y 0.8861, Z 11.0000, A 0.000, B 0.000, C 0.000 }
gfCNCPoint2[6398] = {X 607.6965, Y 0.8861, Z 0.8333, A 0.000, B 0.000, C 0.000 }
gfCNCPoint2[6399] = {X 607.6965, Y 0.8861, Z -2.1667, A 0.000, B 0.000, C 0.000 }
gfCNCPoint2[6400] = {X 603.6965, Y 8.0115, Z -2.1667, A 0.000, B 0.000, C 0.000 }
gfCNCPoint2[6401] = {X 603.2602, Y 8.6459, Z -2.1667, A 0.000, B 0.000, C 0.000 }
gfCNCPoint2[6402] = {X 602.7164, Y 9.1909, Z -2.1667, A 0.000, B 0.000, C 0.000 }
gfCNCPoint2[6403] = {X 602.7163, Y 40.8098, Z -2.1667, A 0.000, B 0.000, C 0.000 }
gfCNCPoint2[6404] = {X 603.2601, Y 41.3546, Z -2.1667, A 0.000, B 0.000, C 0.000 }
gfCNCPoint2[6405] = {X 603.6965, Y 41.9888, Z -2.1667, A 0.000, B 0.000, C 0.000 }
gfCNCPoint2[6406] = {X 607.6965, Y 49.1107, Z -2.1667, A 0.000, B 0.000, C 0.000 }
gfCNCPoint2[6407] = {X 607.6965, Y 49.1107, Z 0.8333, A 0.000, B 0.000, C 0.000 }
gfCNCPoint2[6408] = {X 607.6965, Y 49.1107, Z 11.0000, A 0.000, B 0.000, C 0.000 }
gfCNCPoint2[6409] = {X 607.6950, Y 0.0896, Z 11.0000, A 0.000, B 0.000, C 0.000 }
gfCNCPoint2[6410] = {X 607.6950, Y 0.0896, Z 0.8333, A 0.000, B 0.000, C 0.000 }
gfCNCPoint2[6411] = {X 607.6950, Y 0.0896, Z -2.1667, A 0.000, B 0.000, C 0.000 }
gfCNCPoint2[6412] = {X 603.6965, Y 7.8427, Z -2.1667, A 0.000, B 0.000, C 0.000 }
gfCNCPoint2[6413] = {X 603.2335, Y 8.5522, Z -2.1667, A 0.000, B 0.000, C 0.000 }
gfCNCPoint2[6414] = {X 602.6364, Y 9.1532, Z -2.1667, A 0.000, B 0.000, C 0.000 }
gfCNCPoint2[6415] = {X 602.6363, Y 40.8474, Z -2.1667, A 0.000, B 0.000, C 0.000 }
gfCNCPoint2[6416] = {X 603.2334, Y 41.4482, Z -2.1667, A 0.000, B 0.000, C 0.000 }
gfCNCPoint2[6417] = {X 603.6965, Y 42.1575, Z -2.1667, A 0.000, B 0.000, C 0.000 }
gfCNCPoint2[6418] = {X 607.6965, Y 49.9091, Z -2.1667, A 0.000, B 0.000, C 0.000 }
gfCNCPoint2[6419] = {X 607.6965, Y 49.9091, Z 0.8333, A 0.000, B 0.000, C 0.000 }
gfCNCPoint2[6420] = {X 607.6965, Y 49.9091, Z 11.0000, A 0.000, B 0.000, C 0.000 }
gfCNCPoint2[6421] = {X 607.6538, Y -0.8094, Z 11.0000, A 0.000, B 0.000, C 0.000 }
gfCNCPoint2[6422] = {X 607.6538, Y -0.8094, Z 0.8333, A 0.000, B 0.000, C 0.000 }
gfCNCPoint2[6423] = {X 607.6538, Y -0.8094, Z -2.1667, A 0.000, B 0.000, C 0.000 }
gfCNCPoint2[6424] = {X 603.6965, Y 7.6610, Z -2.1667, A 0.000, B 0.000, C 0.000 }
gfCNCPoint2[6425] = {X 603.2068, Y 8.4565, Z -2.1667, A 0.000, B 0.000, C 0.000 }
gfCNCPoint2[6426] = {X 602.5490, Y 9.1198, Z -2.1667, A 0.000, B 0.000, C 0.000 }
gfCNCPoint2[6427] = {X 602.5564, Y 9.1532, Z -2.1667, A 0.000, B 0.000, C 0.000 }
gfCNCPoint2[6428] = {X 602.5563, Y 40.8855, Z -2.1667, A 0.000, B 0.000, C 0.000 }
gfCNCPoint2[6429] = {X 603.2097, Y 41.5468, Z -2.1667, A 0.000, B 0.000, C 0.000 }
gfCNCPoint2[6430] = {X 603.6965, Y 42.3389, Z -2.1667, A 0.000, B 0.000, C 0.000 }
gfCNCPoint2[6431] = {X 607.6965, Y 50.9050, Z -2.1667, A 0.000, B 0.000, C 0.000 }
gfCNCPoint2[6432] = {X 607.6965, Y 50.9050, Z 0.8333, A 0.000, B 0.000, C 0.000 }
gfCNCPoint2[6433] = {X 607.6965, Y 50.9050, Z 11.0000, A 0.000, B 0.000, C 0.000 }
gfCNCPoint2[6434] = {X 607.4988, Y -1.7337, Z 11.0000, A 0.000, B 0.000, C 0.000 }
gfCNCPoint2[6435] = {X 607.4988, Y -1.7337, Z 0.8333, A 0.000, B 0.000, C 0.000 }
gfCNCPoint2[6436] = {X 607.4988, Y -1.7337, Z -2.1667, A 0.000, B 0.000, C 0.000 }
gfCNCPoint2[6437] = {X 603.6965, Y 7.4625, Z -2.1667, A 0.000, B 0.000, C 0.000 }
gfCNCPoint2[6438] = {X 603.3768, Y 8.0782, Z -2.1667, A 0.000, B 0.000, C 0.000 }
gfCNCPoint2[6439] = {X 602.9556, Y 8.6294, Z -2.1667, A 0.000, B 0.000, C 0.000 }
gfCNCPoint2[6440] = {X 602.4454, Y 9.0995, Z -2.1667, A 0.000, B 0.000, C 0.000 }
gfCNCPoint2[6441] = {X 602.4764, Y 9.1532, Z -2.1667, A 0.000, B 0.000, C 0.000 }
gfCNCPoint2[6442] = {X 602.4763, Y 40.9231, Z -2.1667, A 0.000, B 0.000, C 0.000 }
gfCNCPoint2[6443] = {X 602.5725, Y 41.0029, Z -2.1667, A 0.000, B 0.000, C 0.000 }
gfCNCPoint2[6444] = {X 603.2271, Y 41.7024, Z -2.1667, A 0.000, B 0.000, C 0.000 }
gfCNCPoint2[6445] = {X 603.6965, Y 42.5375, Z -2.1667, A 0.000, B 0.000, C 0.000 }
gfCNCPoint2[6446] = {X 607.6965, Y 52.2117, Z -2.1667, A 0.000, B 0.000, C 0.000 }
gfCNCPoint2[6447] = {X 607.6965, Y 52.2117, Z 0.8333, A 0.000, B 0.000, C 0.000 }
gfCNCPoint2[6448] = {X 607.6965, Y 52.2117, Z 11.0000, A 0.000, B 0.000, C 0.000 }
gfCNCPoint2[6449] = {X 607.6965, Y 2.1252, Z 11.0000, A 0.000, B 0.000, C 0.000 }
gfCNCPoint2[6450] = {X 607.6965, Y 2.1252, Z 0.0000, A 0.000, B 0.000, C 0.000 }
gfCNCPoint2[6451] = {X 607.6965, Y 2.1252, Z -3.0000, A 0.000, B 0.000, C 0.000 }
gfCNCPoint2[6452] = {X 603.6965, Y 8.3206, Z -3.0000, A 0.000, B 0.000, C 0.000 }
gfCNCPoint2[6453] = {X 603.3202, Y 8.8213, Z -3.0000, A 0.000, B 0.000, C 0.000 }
gfCNCPoint2[6454] = {X 602.8767, Y 9.2634, Z -3.0000, A 0.000, B 0.000, C 0.000 }
gfCNCPoint2[6455] = {X 602.8766, Y 40.7365, Z -3.0000, A 0.000, B 0.000, C 0.000 }
gfCNCPoint2[6456] = {X 603.3202, Y 41.1787, Z -3.0000, A 0.000, B 0.000, C 0.000 }
gfCNCPoint2[6457] = {X 603.6965, Y 41.6794, Z -3.0000, A 0.000, B 0.000, C 0.000 }
gfCNCPoint2[6458] = {X 607.6965, Y 47.8749, Z -3.0000, A 0.000, B 0.000, C 0.000 }
gfCNCPoint2[6459] = {X 607.6965, Y 47.8749, Z 0.0000, A 0.000, B 0.000, C 0.000 }
gfCNCPoint2[6460] = {X 607.6965, Y 47.8749, Z 11.0000, A 0.000, B 0.000, C 0.000 }
gfCNCPoint2[6461] = {X 607.6965, Y 1.5504, Z 11.0000, A 0.000, B 0.000, C 0.000 }
gfCNCPoint2[6462] = {X 607.6965, Y 1.5504, Z 0.0000, A 0.000, B 0.000, C 0.000 }
gfCNCPoint2[6463] = {X 607.6965, Y 1.5504, Z -3.0000, A 0.000, B 0.000, C 0.000 }
gfCNCPoint2[6464] = {X 603.6965, Y 8.1705, Z -3.0000, A 0.000, B 0.000, C 0.000 }
gfCNCPoint2[6465] = {X 603.2894, Y 8.7357, Z -3.0000, A 0.000, B 0.000, C 0.000 }
gfCNCPoint2[6466] = {X 602.7967, Y 9.2281, Z -3.0000, A 0.000, B 0.000, C 0.000 }
gfCNCPoint2[6467] = {X 602.7966, Y 40.7726, Z -3.0000, A 0.000, B 0.000, C 0.000 }
gfCNCPoint2[6468] = {X 603.2893, Y 41.2648, Z -3.0000, A 0.000, B 0.000, C 0.000 }
gfCNCPoint2[6469] = {X 603.6965, Y 41.8299, Z -3.0000, A 0.000, B 0.000, C 0.000 }
gfCNCPoint2[6470] = {X 607.6965, Y 48.4470, Z -3.0000, A 0.000, B 0.000, C 0.000 }
gfCNCPoint2[6471] = {X 607.6965, Y 48.4470, Z 0.0000, A 0.000, B 0.000, C 0.000 }
gfCNCPoint2[6472] = {X 607.6965, Y 48.4470, Z 11.0000, A 0.000, B 0.000, C 0.000 }
gfCNCPoint2[6473] = {X 607.6965, Y 0.8845, Z 11.0000, A 0.000, B 0.000, C 0.000 }
gfCNCPoint2[6474] = {X 607.6965, Y 0.8845, Z 0.0000, A 0.000, B 0.000, C 0.000 }
gfCNCPoint2[6475] = {X 607.6965, Y 0.8845, Z -3.0000, A 0.000, B 0.000, C 0.000 }
gfCNCPoint2[6476] = {X 603.6965, Y 8.0115, Z -3.0000, A 0.000, B 0.000, C 0.000 }
gfCNCPoint2[6477] = {X 603.2604, Y 8.6459, Z -3.0000, A 0.000, B 0.000, C 0.000 }
gfCNCPoint2[6478] = {X 602.7167, Y 9.1909, Z -3.0000, A 0.000, B 0.000, C 0.000 }
gfCNCPoint2[6479] = {X 602.7166, Y 40.8098, Z -3.0000, A 0.000, B 0.000, C 0.000 }
gfCNCPoint2[6480] = {X 603.2603, Y 41.3546, Z -3.0000, A 0.000, B 0.000, C 0.000 }
gfCNCPoint2[6481] = {X 603.6965, Y 41.9887, Z -3.0000, A 0.000, B 0.000, C 0.000 }
gfCNCPoint2[6482] = {X 607.6965, Y 49.1122, Z -3.0000, A 0.000, B 0.000, C 0.000 }
gfCNCPoint2[6483] = {X 607.6965, Y 49.1122, Z 0.0000, A 0.000, B 0.000, C 0.000 }
gfCNCPoint2[6484] = {X 607.6965, Y 49.1122, Z 11.0000, A 0.000, B 0.000, C 0.000 }
gfCNCPoint2[6485] = {X 607.6950, Y 0.0877, Z 11.0000, A 0.000, B 0.000, C 0.000 }
gfCNCPoint2[6486] = {X 607.6950, Y 0.0877, Z 0.0000, A 0.000, B 0.000, C 0.000 }
gfCNCPoint2[6487] = {X 607.6950, Y 0.0877, Z -3.0000, A 0.000, B 0.000, C 0.000 }
gfCNCPoint2[6488] = {X 603.6965, Y 7.8428, Z -3.0000, A 0.000, B 0.000, C 0.000 }
gfCNCPoint2[6489] = {X 603.2337, Y 8.5522, Z -3.0000, A 0.000, B 0.000, C 0.000 }
gfCNCPoint2[6490] = {X 602.6367, Y 9.1532, Z -3.0000, A 0.000, B 0.000, C 0.000 }
gfCNCPoint2[6491] = {X 602.6366, Y 40.8474, Z -3.0000, A 0.000, B 0.000, C 0.000 }
gfCNCPoint2[6492] = {X 603.2336, Y 41.4482, Z -3.0000, A 0.000, B 0.000, C 0.000 }
gfCNCPoint2[6493] = {X 603.6965, Y 42.1575, Z -3.0000, A 0.000, B 0.000, C 0.000 }
gfCNCPoint2[6494] = {X 607.6965, Y 49.9110, Z -3.0000, A 0.000, B 0.000, C 0.000 }
gfCNCPoint2[6495] = {X 607.6965, Y 49.9110, Z 0.0000, A 0.000, B 0.000, C 0.000 }
gfCNCPoint2[6496] = {X 607.6965, Y 49.9110, Z 11.0000, A 0.000, B 0.000, C 0.000 }
gfCNCPoint2[6497] = {X 607.6538, Y -0.8098, Z 11.0000, A 0.000, B 0.000, C 0.000 }
gfCNCPoint2[6498] = {X 607.6538, Y -0.8098, Z 0.0000, A 0.000, B 0.000, C 0.000 }
gfCNCPoint2[6499] = {X 607.6538, Y -0.8098, Z -3.0000, A 0.000, B 0.000, C 0.000 }
gfCNCPoint2[6500] = {X 603.6965, Y 7.6610, Z -3.0000, A 0.000, B 0.000, C 0.000 }
gfCNCPoint2[6501] = {X 603.2069, Y 8.4564, Z -3.0000, A 0.000, B 0.000, C 0.000 }
gfCNCPoint2[6502] = {X 602.5493, Y 9.1196, Z -3.0000, A 0.000, B 0.000, C 0.000 }
gfCNCPoint2[6503] = {X 602.5567, Y 9.1532, Z -3.0000, A 0.000, B 0.000, C 0.000 }
gfCNCPoint2[6504] = {X 602.5566, Y 40.8855, Z -3.0000, A 0.000, B 0.000, C 0.000 }
gfCNCPoint2[6505] = {X 603.2099, Y 41.5468, Z -3.0000, A 0.000, B 0.000, C 0.000 }
gfCNCPoint2[6506] = {X 603.6965, Y 42.3389, Z -3.0000, A 0.000, B 0.000, C 0.000 }
gfCNCPoint2[6507] = {X 607.6965, Y 50.9076, Z -3.0000, A 0.000, B 0.000, C 0.000 }
gfCNCPoint2[6508] = {X 607.6965, Y 50.9076, Z 0.0000, A 0.000, B 0.000, C 0.000 }
gfCNCPoint2[6509] = {X 607.6965, Y 50.9076, Z 11.0000, A 0.000, B 0.000, C 0.000 }
gfCNCPoint2[6510] = {X 607.4988, Y -1.7340, Z 11.0000, A 0.000, B 0.000, C 0.000 }
gfCNCPoint2[6511] = {X 607.4988, Y -1.7340, Z 0.0000, A 0.000, B 0.000, C 0.000 }
gfCNCPoint2[6512] = {X 607.4988, Y -1.7340, Z -3.0000, A 0.000, B 0.000, C 0.000 }
gfCNCPoint2[6513] = {X 603.6965, Y 7.4624, Z -3.0000, A 0.000, B 0.000, C 0.000 }
gfCNCPoint2[6514] = {X 603.3768, Y 8.0781, Z -3.0000, A 0.000, B 0.000, C 0.000 }
gfCNCPoint2[6515] = {X 602.9556, Y 8.6293, Z -3.0000, A 0.000, B 0.000, C 0.000 }
gfCNCPoint2[6516] = {X 602.4454, Y 9.0995, Z -3.0000, A 0.000, B 0.000, C 0.000 }
gfCNCPoint2[6517] = {X 602.4767, Y 9.1532, Z -3.0000, A 0.000, B 0.000, C 0.000 }
gfCNCPoint2[6518] = {X 602.4766, Y 40.9230, Z -3.0000, A 0.000, B 0.000, C 0.000 }
gfCNCPoint2[6519] = {X 602.5726, Y 41.0030, Z -3.0000, A 0.000, B 0.000, C 0.000 }
gfCNCPoint2[6520] = {X 603.2271, Y 41.7025, Z -3.0000, A 0.000, B 0.000, C 0.000 }
gfCNCPoint2[6521] = {X 603.6965, Y 42.5376, Z -3.0000, A 0.000, B 0.000, C 0.000 }
gfCNCPoint2[6522] = {X 607.6965, Y 52.2123, Z -3.0000, A 0.000, B 0.000, C 0.000 }
gfCNCPoint2[6523] = {X 607.6965, Y 52.2123, Z 0.0000, A 0.000, B 0.000, C 0.000 }
gfCNCPoint2[6524] = {X 607.6965, Y 52.2123, Z 11.0000, A 0.000, B 0.000, C 0.000 }
gfCNCPoint2[6525] = {X 492.1943, Y 19.7812, Z 11.0000, A 0.000, B 0.000, C 0.000 }
gfCNCPoint2[6526] = {X 492.1943, Y 19.7812, Z 0.8333, A 0.000, B 0.000, C 0.000 }
gfCNCPoint2[6527] = {X 487.6645, Y 19.7804, Z -0.3804, A 0.000, B 0.000, C 0.000 }
gfCNCPoint2[6528] = {X 486.9699, Y 19.7851, Z -0.5666, A 0.000, B 0.000, C 0.000 }
gfCNCPoint2[6529] = {X 486.2675, Y 19.7837, Z -0.7548, A 0.000, B 0.000, C 0.000 }
gfCNCPoint2[6530] = {X 485.4758, Y 19.8887, Z -0.9688, A 0.000, B 0.000, C 0.000 }
gfCNCPoint2[6531] = {X 484.7981, Y 20.0732, Z -1.1570, A 0.000, B 0.000, C 0.000 }
gfCNCPoint2[6532] = {X 484.6640, Y 20.1097, Z -1.1942, A 0.000, B 0.000, C 0.000 }
gfCNCPoint2[6533] = {X 484.6328, Y 20.1389, Z -1.2056, A 0.000, B 0.000, C 0.000 }
gfCNCPoint2[6534] = {X 484.5881, Y 20.2705, Z -1.2429, A 0.000, B 0.000, C 0.000 }
gfCNCPoint2[6535] = {X 484.4392, Y 20.7081, Z -1.3667, A 0.000, B 0.000, C 0.000 }
gfCNCPoint2[6536] = {X 484.4037, Y 21.9094, Z -1.6888, A 0.000, B 0.000, C 0.000 }
gfCNCPoint2[6537] = {X 484.5265, Y 22.3550, Z -1.8126, A 0.000, B 0.000, C 0.000 }
gfCNCPoint2[6538] = {X 484.6986, Y 22.4110, Z -1.8611, A 0.000, B 0.000, C 0.000 }
gfCNCPoint2[6539] = {X 484.8786, Y 22.4308, Z -1.9096, A 0.000, B 0.000, C 0.000 }
gfCNCPoint2[6540] = {X 486.0431, Y 22.5560, Z -2.2235, A 0.000, B 0.000, C 0.000 }
gfCNCPoint2[6541] = {X 487.1636, Y 22.5560, Z -2.5237, A 0.000, B 0.000, C 0.000 }
gfCNCPoint2[6542] = {X 488.9411, Y 22.5560, Z -3.0000, A 0.000, B 0.000, C 0.000 }
gfCNCPoint2[6543] = {X 493.3690, Y 22.5560, Z -3.0000, A 0.000, B 0.000, C 0.000 }
gfCNCPoint2[6544] = {X 493.3690, Y 19.7814, Z -3.0000, A 0.000, B 0.000, C 0.000 }
gfCNCPoint2[6545] = {X 487.6645, Y 19.7804, Z -3.0000, A 0.000, B 0.000, C 0.000 }
gfCNCPoint2[6546] = {X 486.9699, Y 19.7851, Z -3.0000, A 0.000, B 0.000, C 0.000 }
gfCNCPoint2[6547] = {X 485.8743, Y 19.8564, Z -3.0000, A 0.000, B 0.000, C 0.000 }
gfCNCPoint2[6548] = {X 484.7981, Y 20.0732, Z -3.0000, A 0.000, B 0.000, C 0.000 }
gfCNCPoint2[6549] = {X 484.6685, Y 20.1457, Z -3.0000, A 0.000, B 0.000, C 0.000 }
gfCNCPoint2[6550] = {X 484.5881, Y 20.2705, Z -3.0000, A 0.000, B 0.000, C 0.000 }
gfCNCPoint2[6551] = {X 484.4285, Y 20.9566, Z -3.0000, A 0.000, B 0.000, C 0.000 }
gfCNCPoint2[6552] = {X 484.4077, Y 21.6607, Z -3.0000, A 0.000, B 0.000, C 0.000 }
gfCNCPoint2[6553] = {X 484.5265, Y 22.3550, Z -3.0000, A 0.000, B 0.000, C 0.000 }
gfCNCPoint2[6554] = {X 484.7006, Y 22.4019, Z -3.0000, A 0.000, B 0.000, C 0.000 }
gfCNCPoint2[6555] = {X 484.8786, Y 22.4308, Z -3.0000, A 0.000, B 0.000, C 0.000 }
gfCNCPoint2[6556] = {X 486.0194, Y 22.5247, Z -3.0000, A 0.000, B 0.000, C 0.000 }
gfCNCPoint2[6557] = {X 487.1636, Y 22.5560, Z -3.0000, A 0.000, B 0.000, C 0.000 }
gfCNCPoint2[6558] = {X 488.9411, Y 22.5560, Z -3.0000, A 0.000, B 0.000, C 0.000 }
gfCNCPoint2[6559] = {X 484.9563, Y 22.2874, Z -3.0000, A 0.000, B 0.000, C 0.000 }
gfCNCPoint2[6560] = {X 488.9411, Y 22.6360, Z -3.0000, A 0.000, B 0.000, C 0.000 }
gfCNCPoint2[6561] = {X 493.4490, Y 22.6360, Z -3.0000, A 0.000, B 0.000, C 0.000 }
gfCNCPoint2[6562] = {X 493.4490, Y 19.7014, Z -3.0000, A 0.000, B 0.000, C 0.000 }
gfCNCPoint2[6563] = {X 487.6642, Y 19.7004, Z -3.0000, A 0.000, B 0.000, C 0.000 }
gfCNCPoint2[6564] = {X 486.9714, Y 19.7052, Z -3.0000, A 0.000, B 0.000, C 0.000 }
gfCNCPoint2[6565] = {X 485.8645, Y 19.7770, Z -3.0000, A 0.000, B 0.000, C 0.000 }
gfCNCPoint2[6566] = {X 484.7771, Y 19.9960, Z -3.0000, A 0.000, B 0.000, C 0.000 }
gfCNCPoint2[6567] = {X 484.6137, Y 20.0874, Z -3.0000, A 0.000, B 0.000, C 0.000 }
gfCNCPoint2[6568] = {X 484.5123, Y 20.2447, Z -3.0000, A 0.000, B 0.000, C 0.000 }
gfCNCPoint2[6569] = {X 484.3474, Y 20.9604, Z -3.0000, A 0.000, B 0.000, C 0.000 }
gfCNCPoint2[6570] = {X 484.3300, Y 21.6946, Z -3.0000, A 0.000, B 0.000, C 0.000 }
gfCNCPoint2[6571] = {X 484.4609, Y 22.4173, Z -3.0000, A 0.000, B 0.000, C 0.000 }
gfCNCPoint2[6572] = {X 484.6627, Y 22.4755, Z -3.0000, A 0.000, B 0.000, C 0.000 }
gfCNCPoint2[6573] = {X 484.8698, Y 22.5103, Z -3.0000, A 0.000, B 0.000, C 0.000 }
gfCNCPoint2[6574] = {X 486.0150, Y 22.6046, Z -3.0000, A 0.000, B 0.000, C 0.000 }
gfCNCPoint2[6575] = {X 487.1636, Y 22.6360, Z -3.0000, A 0.000, B 0.000, C 0.000 }
gfCNCPoint2[6576] = {X 488.9411, Y 22.6360, Z -3.0000, A 0.000, B 0.000, C 0.000 }
gfCNCPoint2[6577] = {X 492.9259, Y 22.2874, Z -3.0000, A 0.000, B 0.000, C 0.000 }
gfCNCPoint2[6578] = {X 484.9563, Y 22.3674, Z -3.0000, A 0.000, B 0.000, C 0.000 }
gfCNCPoint2[6579] = {X 488.9411, Y 22.7160, Z -3.0000, A 0.000, B 0.000, C 0.000 }
gfCNCPoint2[6580] = {X 493.5290, Y 22.7160, Z -3.0000, A 0.000, B 0.000, C 0.000 }
gfCNCPoint2[6581] = {X 493.5290, Y 19.6214, Z -3.0000, A 0.000, B 0.000, C 0.000 }
gfCNCPoint2[6582] = {X 487.6640, Y 19.6204, Z -3.0000, A 0.000, B 0.000, C 0.000 }
gfCNCPoint2[6583] = {X 486.9712, Y 19.6252, Z -3.0000, A 0.000, B 0.000, C 0.000 }
gfCNCPoint2[6584] = {X 485.8538, Y 19.6977, Z -3.0000, A 0.000, B 0.000, C 0.000 }
gfCNCPoint2[6585] = {X 484.7560, Y 19.9188, Z -3.0000, A 0.000, B 0.000, C 0.000 }
gfCNCPoint2[6586] = {X 484.5589, Y 20.0291, Z -3.0000, A 0.000, B 0.000, C 0.000 }
gfCNCPoint2[6587] = {X 484.4366, Y 20.2190, Z -3.0000, A 0.000, B 0.000, C 0.000 }
gfCNCPoint2[6588] = {X 484.2664, Y 20.9639, Z -3.0000, A 0.000, B 0.000, C 0.000 }
gfCNCPoint2[6589] = {X 484.2525, Y 21.7280, Z -3.0000, A 0.000, B 0.000, C 0.000 }
gfCNCPoint2[6590] = {X 484.3956, Y 22.4786, Z -3.0000, A 0.000, B 0.000, C 0.000 }
gfCNCPoint2[6591] = {X 484.6249, Y 22.5488, Z -3.0000, A 0.000, B 0.000, C 0.000 }
gfCNCPoint2[6592] = {X 484.8611, Y 22.5898, Z -3.0000, A 0.000, B 0.000, C 0.000 }
gfCNCPoint2[6593] = {X 486.0106, Y 22.6845, Z -3.0000, A 0.000, B 0.000, C 0.000 }
gfCNCPoint2[6594] = {X 487.1636, Y 22.7160, Z -3.0000, A 0.000, B 0.000, C 0.000 }
gfCNCPoint2[6595] = {X 488.9411, Y 22.7160, Z -3.0000, A 0.000, B 0.000, C 0.000 }
gfCNCPoint2[6596] = {X 492.9259, Y 22.3674, Z -3.0000, A 0.000, B 0.000, C 0.000 }
gfCNCPoint2[6597] = {X 484.9563, Y 22.4474, Z -3.0000, A 0.000, B 0.000, C 0.000 }
gfCNCPoint2[6598] = {X 488.9411, Y 22.7960, Z -3.0000, A 0.000, B 0.000, C 0.000 }
gfCNCPoint2[6599] = {X 493.6090, Y 22.7960, Z -3.0000, A 0.000, B 0.000, C 0.000 }
gfCNCPoint2[6600] = {X 493.6090, Y 19.5414, Z -3.0000, A 0.000, B 0.000, C 0.000 }
gfCNCPoint2[6601] = {X 487.6637, Y 19.5404, Z -3.0000, A 0.000, B 0.000, C 0.000 }
gfCNCPoint2[6602] = {X 486.9711, Y 19.5451, Z -3.0000, A 0.000, B 0.000, C 0.000 }
gfCNCPoint2[6603] = {X 485.8431, Y 19.6184, Z -3.0000, A 0.000, B 0.000, C 0.000 }
gfCNCPoint2[6604] = {X 484.7350, Y 19.8416, Z -3.0000, A 0.000, B 0.000, C 0.000 }
gfCNCPoint2[6605] = {X 484.5041, Y 19.9708, Z -3.0000, A 0.000, B 0.000, C 0.000 }
gfCNCPoint2[6606] = {X 484.3609, Y 20.1932, Z -3.0000, A 0.000, B 0.000, C 0.000 }
gfCNCPoint2[6607] = {X 484.1854, Y 20.9672, Z -3.0000, A 0.000, B 0.000, C 0.000 }
gfCNCPoint2[6608] = {X 484.1751, Y 21.7609, Z -3.0000, A 0.000, B 0.000, C 0.000 }
gfCNCPoint2[6609] = {X 484.3305, Y 22.5392, Z -3.0000, A 0.000, B 0.000, C 0.000 }
gfCNCPoint2[6610] = {X 484.5870, Y 22.6219, Z -3.0000, A 0.000, B 0.000, C 0.000 }
gfCNCPoint2[6611] = {X 484.8523, Y 22.6694, Z -3.0000, A 0.000, B 0.000, C 0.000 }
gfCNCPoint2[6612] = {X 486.0062, Y 22.7644, Z -3.0000, A 0.000, B 0.000, C 0.000 }
gfCNCPoint2[6613] = {X 487.1636, Y 22.7960, Z -3.0000, A 0.000, B 0.000, C 0.000 }
gfCNCPoint2[6614] = {X 488.9411, Y 22.7960, Z -3.0000, A 0.000, B 0.000, C 0.000 }
gfCNCPoint2[6615] = {X 492.9259, Y 22.4474, Z -3.0000, A 0.000, B 0.000, C 0.000 }
gfCNCPoint2[6616] = {X 484.9563, Y 22.5274, Z -3.0000, A 0.000, B 0.000, C 0.000 }
gfCNCPoint2[6617] = {X 488.9411, Y 22.8760, Z -3.0000, A 0.000, B 0.000, C 0.000 }
gfCNCPoint2[6618] = {X 493.6890, Y 22.8760, Z -3.0000, A 0.000, B 0.000, C 0.000 }
gfCNCPoint2[6619] = {X 493.6890, Y 19.4614, Z -3.0000, A 0.000, B 0.000, C 0.000 }
gfCNCPoint2[6620] = {X 487.6634, Y 19.4604, Z -3.0000, A 0.000, B 0.000, C 0.000 }
gfCNCPoint2[6621] = {X 486.9709, Y 19.4651, Z -3.0000, A 0.000, B 0.000, C 0.000 }
gfCNCPoint2[6622] = {X 485.8324, Y 19.5391, Z -3.0000, A 0.000, B 0.000, C 0.000 }
gfCNCPoint2[6623] = {X 484.7140, Y 19.7644, Z -3.0000, A 0.000, B 0.000, C 0.000 }
gfCNCPoint2[6624] = {X 484.4494, Y 19.9125, Z -3.0000, A 0.000, B 0.000, C 0.000 }
gfCNCPoint2[6625] = {X 484.2851, Y 20.1674, Z -3.0000, A 0.000, B 0.000, C 0.000 }
gfCNCPoint2[6626] = {X 484.1045, Y 20.9703, Z -3.0000, A 0.000, B 0.000, C 0.000 }
gfCNCPoint2[6627] = {X 484.0978, Y 21.7933, Z -3.0000, A 0.000, B 0.000, C 0.000 }
gfCNCPoint2[6628] = {X 484.2655, Y 22.5990, Z -3.0000, A 0.000, B 0.000, C 0.000 }
gfCNCPoint2[6629] = {X 484.5491, Y 22.6948, Z -3.0000, A 0.000, B 0.000, C 0.000 }
gfCNCPoint2[6630] = {X 484.8436, Y 22.7489, Z -3.0000, A 0.000, B 0.000, C 0.000 }
gfCNCPoint2[6631] = {X 486.0018, Y 22.8442, Z -3.0000, A 0.000, B 0.000, C 0.000 }
gfCNCPoint2[6632] = {X 487.1636, Y 22.8760, Z -3.0000, A 0.000, B 0.000, C 0.000 }
gfCNCPoint2[6633] = {X 488.9411, Y 22.8760, Z -3.0000, A 0.000, B 0.000, C 0.000 }
gfCNCPoint2[6634] = {X 492.9259, Y 22.5274, Z -3.0000, A 0.000, B 0.000, C 0.000 }
gfCNCPoint2[6635] = {X 484.9563, Y 22.6074, Z -3.0000, A 0.000, B 0.000, C 0.000 }
gfCNCPoint2[6636] = {X 488.9411, Y 22.9560, Z -3.0000, A 0.000, B 0.000, C 0.000 }
gfCNCPoint2[6637] = {X 493.7690, Y 22.9560, Z -3.0000, A 0.000, B 0.000, C 0.000 }
gfCNCPoint2[6638] = {X 493.7700, Y 19.3814, Z -3.0000, A 0.000, B 0.000, C 0.000 }
gfCNCPoint2[6639] = {X 487.6632, Y 19.3804, Z -3.0000, A 0.000, B 0.000, C 0.000 }
gfCNCPoint2[6640] = {X 486.9707, Y 19.3851, Z -3.0000, A 0.000, B 0.000, C 0.000 }
gfCNCPoint2[6641] = {X 485.8217, Y 19.4598, Z -3.0000, A 0.000, B 0.000, C 0.000 }
gfCNCPoint2[6642] = {X 484.6930, Y 19.6872, Z -3.0000, A 0.000, B 0.000, C 0.000 }
gfCNCPoint2[6643] = {X 484.3946, Y 19.8542, Z -3.0000, A 0.000, B 0.000, C 0.000 }
gfCNCPoint2[6644] = {X 484.2094, Y 20.1416, Z -3.0000, A 0.000, B 0.000, C 0.000 }
gfCNCPoint2[6645] = {X 484.0236, Y 20.9733, Z -3.0000, A 0.000, B 0.000, C 0.000 }
gfCNCPoint2[6646] = {X 484.0207, Y 21.8254, Z -3.0000, A 0.000, B 0.000, C 0.000 }
gfCNCPoint2[6647] = {X 484.2007, Y 22.6582, Z -3.0000, A 0.000, B 0.000, C 0.000 }
gfCNCPoint2[6648] = {X 484.5113, Y 22.7676, Z -3.0000, A 0.000, B 0.000, C 0.000 }
gfCNCPoint2[6649] = {X 484.8349, Y 22.8284, Z -3.0000, A 0.000, B 0.000, C 0.000 }
gfCNCPoint2[6650] = {X 485.9975, Y 22.9241, Z -3.0000, A 0.000, B 0.000, C 0.000 }
gfCNCPoint2[6651] = {X 487.1636, Y 22.9560, Z -3.0000, A 0.000, B 0.000, C 0.000 }
gfCNCPoint2[6652] = {X 488.9411, Y 22.9560, Z -3.0000, A 0.000, B 0.000, C 0.000 }
gfCNCPoint2[6653] = {X 492.9259, Y 22.6074, Z -3.0000, A 0.000, B 0.000, C 0.000 }
gfCNCPoint2[6654] = {X 492.9259, Y 22.6074, Z 0.0000, A 0.000, B 0.000, C 0.000 }
gfCNCPoint2[6655] = {X 492.9259, Y 22.6074, Z 11.0000, A 0.000, B 0.000, C 0.000 }
gfCNCPoint2[6656] = {X 448.7124, Y 19.7813, Z 11.0000, A 0.000, B 0.000, C 0.000 }
gfCNCPoint2[6657] = {X 448.7124, Y 19.7813, Z 0.8333, A 0.000, B 0.000, C 0.000 }
gfCNCPoint2[6658] = {X 444.0413, Y 19.7811, Z -0.4183, A 0.000, B 0.000, C 0.000 }
gfCNCPoint2[6659] = {X 443.3489, Y 19.7973, Z -0.6039, A 0.000, B 0.000, C 0.000 }
gfCNCPoint2[6660] = {X 442.7483, Y 19.8043, Z -0.7648, A 0.000, B 0.000, C 0.000 }
gfCNCPoint2[6661] = {X 442.0370, Y 19.9275, Z -0.9582, A 0.000, B 0.000, C 0.000 }
gfCNCPoint2[6662] = {X 441.4690, Y 20.1228, Z -1.1192, A 0.000, B 0.000, C 0.000 }
gfCNCPoint2[6663] = {X 441.3661, Y 20.1582, Z -1.1483, A 0.000, B 0.000, C 0.000 }
gfCNCPoint2[6664] = {X 441.1882, Y 20.7176, Z -1.3056, A 0.000, B 0.000, C 0.000 }
gfCNCPoint2[6665] = {X 441.1544, Y 21.8888, Z -1.6196, A 0.000, B 0.000, C 0.000 }
gfCNCPoint2[6666] = {X 441.2728, Y 22.3520, Z -1.7477, A 0.000, B 0.000, C 0.000 }
gfCNCPoint2[6667] = {X 441.5016, Y 22.4268, Z -1.8122, A 0.000, B 0.000, C 0.000 }
gfCNCPoint2[6668] = {X 441.7413, Y 22.4488, Z -1.8767, A 0.000, B 0.000, C 0.000 }
gfCNCPoint2[6669] = {X 442.9870, Y 22.5629, Z -2.2118, A 0.000, B 0.000, C 0.000 }
gfCNCPoint2[6670] = {X 443.1393, Y 22.5691, Z -2.2527, A 0.000, B 0.000, C 0.000 }
gfCNCPoint2[6671] = {X 444.3942, Y 22.5560, Z -2.5890, A 0.000, B 0.000, C 0.000 }
gfCNCPoint2[6672] = {X 445.9282, Y 22.5560, Z -3.0000, A 0.000, B 0.000, C 0.000 }
gfCNCPoint2[6673] = {X 450.1184, Y 22.5560, Z -3.0000, A 0.000, B 0.000, C 0.000 }
gfCNCPoint2[6674] = {X 450.1184, Y 19.7814, Z -3.0000, A 0.000, B 0.000, C 0.000 }
gfCNCPoint2[6675] = {X 444.0413, Y 19.7811, Z -3.0000, A 0.000, B 0.000, C 0.000 }
gfCNCPoint2[6676] = {X 443.3489, Y 19.7973, Z -3.0000, A 0.000, B 0.000, C 0.000 }
gfCNCPoint2[6677] = {X 442.3959, Y 19.8848, Z -3.0000, A 0.000, B 0.000, C 0.000 }
gfCNCPoint2[6678] = {X 441.4690, Y 20.1228, Z -3.0000, A 0.000, B 0.000, C 0.000 }
gfCNCPoint2[6679] = {X 441.3845, Y 20.1762, Z -3.0000, A 0.000, B 0.000, C 0.000 }
gfCNCPoint2[6680] = {X 441.3331, Y 20.2620, Z -3.0000, A 0.000, B 0.000, C 0.000 }
gfCNCPoint2[6681] = {X 441.1827, Y 20.9508, Z -3.0000, A 0.000, B 0.000, C 0.000 }
gfCNCPoint2[6682] = {X 441.1624, Y 21.6556, Z -3.0000, A 0.000, B 0.000, C 0.000 }
gfCNCPoint2[6683] = {X 441.2728, Y 22.3520, Z -3.0000, A 0.000, B 0.000, C 0.000 }
gfCNCPoint2[6684] = {X 441.5044, Y 22.4136, Z -3.0000, A 0.000, B 0.000, C 0.000 }
gfCNCPoint2[6685] = {X 441.7413, Y 22.4488, Z -3.0000, A 0.000, B 0.000, C 0.000 }
gfCNCPoint2[6686] = {X 443.0664, Y 22.5362, Z -3.0000, A 0.000, B 0.000, C 0.000 }
gfCNCPoint2[6687] = {X 444.3942, Y 22.5560, Z -3.0000, A 0.000, B 0.000, C 0.000 }
gfCNCPoint2[6688] = {X 445.9282, Y 22.5560, Z -3.0000, A 0.000, B 0.000, C 0.000 }
gfCNCPoint2[6689] = {X 441.9435, Y 22.2874, Z -3.0000, A 0.000, B 0.000, C 0.000 }
gfCNCPoint2[6690] = {X 445.9282, Y 22.6360, Z -3.0000, A 0.000, B 0.000, C 0.000 }
gfCNCPoint2[6691] = {X 450.1984, Y 22.6360, Z -3.0000, A 0.000, B 0.000, C 0.000 }
gfCNCPoint2[6692] = {X 450.1984, Y 19.7014, Z -3.0000, A 0.000, B 0.000, C 0.000 }
gfCNCPoint2[6693] = {X 444.0404, Y 19.7011, Z -3.0000, A 0.000, B 0.000, C 0.000 }
gfCNCPoint2[6694] = {X 443.3498, Y 19.7173, Z -3.0000, A 0.000, B 0.000, C 0.000 }
gfCNCPoint2[6695] = {X 442.3832, Y 19.8058, Z -3.0000, A 0.000, B 0.000, C 0.000 }
gfCNCPoint2[6696] = {X 441.4430, Y 20.0471, Z -3.0000, A 0.000, B 0.000, C 0.000 }
gfCNCPoint2[6697] = {X 441.3273, Y 20.1203, Z -3.0000, A 0.000, B 0.000, C 0.000 }
gfCNCPoint2[6698] = {X 441.2568, Y 20.2377, Z -3.0000, A 0.000, B 0.000, C 0.000 }
gfCNCPoint2[6699] = {X 441.1016, Y 20.9555, Z -3.0000, A 0.000, B 0.000, C 0.000 }
gfCNCPoint2[6700] = {X 441.0845, Y 21.6897, Z -3.0000, A 0.000, B 0.000, C 0.000 }
gfCNCPoint2[6701] = {X 441.2064, Y 22.4139, Z -3.0000, A 0.000, B 0.000, C 0.000 }
gfCNCPoint2[6702] = {X 441.4667, Y 22.4873, Z -3.0000, A 0.000, B 0.000, C 0.000 }
gfCNCPoint2[6703] = {X 441.7340, Y 22.5284, Z -3.0000, A 0.000, B 0.000, C 0.000 }
gfCNCPoint2[6704] = {X 443.0619, Y 22.6161, Z -3.0000, A 0.000, B 0.000, C 0.000 }
gfCNCPoint2[6705] = {X 444.3926, Y 22.6360, Z -3.0000, A 0.000, B 0.000, C 0.000 }
gfCNCPoint2[6706] = {X 445.9282, Y 22.6360, Z -3.0000, A 0.000, B 0.000, C 0.000 }
gfCNCPoint2[6707] = {X 449.9130, Y 22.2874, Z -3.0000, A 0.000, B 0.000, C 0.000 }
gfCNCPoint2[6708] = {X 441.9435, Y 22.3674, Z -3.0000, A 0.000, B 0.000, C 0.000 }
gfCNCPoint2[6709] = {X 445.9282, Y 22.7160, Z -3.0000, A 0.000, B 0.000, C 0.000 }
gfCNCPoint2[6710] = {X 450.2784, Y 22.7160, Z -3.0000, A 0.000, B 0.000, C 0.000 }
gfCNCPoint2[6711] = {X 450.2784, Y 19.6214, Z -3.0000, A 0.000, B 0.000, C 0.000 }
gfCNCPoint2[6712] = {X 444.0395, Y 19.6211, Z -3.0000, A 0.000, B 0.000, C 0.000 }
gfCNCPoint2[6713] = {X 443.3484, Y 19.6373, Z -3.0000, A 0.000, B 0.000, C 0.000 }
gfCNCPoint2[6714] = {X 442.3693, Y 19.7270, Z -3.0000, A 0.000, B 0.000, C 0.000 }
gfCNCPoint2[6715] = {X 441.4170, Y 19.9715, Z -3.0000, A 0.000, B 0.000, C 0.000 }
gfCNCPoint2[6716] = {X 441.2701, Y 20.0644, Z -3.0000, A 0.000, B 0.000, C 0.000 }
gfCNCPoint2[6717] = {X 441.1806, Y 20.2135, Z -3.0000, A 0.000, B 0.000, C 0.000 }
gfCNCPoint2[6718] = {X 441.0205, Y 20.9600, Z -3.0000, A 0.000, B 0.000, C 0.000 }
gfCNCPoint2[6719] = {X 441.0069, Y 21.7234, Z -3.0000, A 0.000, B 0.000, C 0.000 }
gfCNCPoint2[6720] = {X 441.1402, Y 22.4751, Z -3.0000, A 0.000, B 0.000, C 0.000 }
gfCNCPoint2[6721] = {X 441.4291, Y 22.5609, Z -3.0000, A 0.000, B 0.000, C 0.000 }
gfCNCPoint2[6722] = {X 441.7267, Y 22.6081, Z -3.0000, A 0.000, B 0.000, C 0.000 }
gfCNCPoint2[6723] = {X 443.0585, Y 22.6960, Z -3.0000, A 0.000, B 0.000, C 0.000 }
gfCNCPoint2[6724] = {X 444.3930, Y 22.7160, Z -3.0000, A 0.000, B 0.000, C 0.000 }
gfCNCPoint2[6725] = {X 445.9282, Y 22.7160, Z -3.0000, A 0.000, B 0.000, C 0.000 }
gfCNCPoint2[6726] = {X 449.9130, Y 22.3674, Z -3.0000, A 0.000, B 0.000, C 0.000 }
gfCNCPoint2[6727] = {X 441.9435, Y 22.4474, Z -3.0000, A 0.000, B 0.000, C 0.000 }
gfCNCPoint2[6728] = {X 445.9282, Y 22.7960, Z -3.0000, A 0.000, B 0.000, C 0.000 }
gfCNCPoint2[6729] = {X 450.3584, Y 22.7960, Z -3.0000, A 0.000, B 0.000, C 0.000 }
gfCNCPoint2[6730] = {X 450.3584, Y 19.5414, Z -3.0000, A 0.000, B 0.000, C 0.000 }
gfCNCPoint2[6731] = {X 444.0385, Y 19.5411, Z -3.0000, A 0.000, B 0.000, C 0.000 }
gfCNCPoint2[6732] = {X 443.3470, Y 19.5573, Z -3.0000, A 0.000, B 0.000, C 0.000 }
gfCNCPoint2[6733] = {X 442.3554, Y 19.6482, Z -3.0000, A 0.000, B 0.000, C 0.000 }
gfCNCPoint2[6734] = {X 441.3910, Y 19.8958, Z -3.0000, A 0.000, B 0.000, C 0.000 }
gfCNCPoint2[6735] = {X 441.2129, Y 20.0085, Z -3.0000, A 0.000, B 0.000, C 0.000 }
gfCNCPoint2[6736] = {X 441.1044, Y 20.1892, Z -3.0000, A 0.000, B 0.000, C 0.000 }
gfCNCPoint2[6737] = {X 440.9395, Y 20.9643, Z -3.0000, A 0.000, B 0.000, C 0.000 }
gfCNCPoint2[6738] = {X 440.9293, Y 21.7566, Z -3.0000, A 0.000, B 0.000, C 0.000 }
gfCNCPoint2[6739] = {X 441.0742, Y 22.5356, Z -3.0000, A 0.000, B 0.000, C 0.000 }
gfCNCPoint2[6740] = {X 441.3915, Y 22.6344, Z -3.0000, A 0.000, B 0.000, C 0.000 }
gfCNCPoint2[6741] = {X 441.7194, Y 22.6878, Z -3.0000, A 0.000, B 0.000, C 0.000 }
gfCNCPoint2[6742] = {X 443.0550, Y 22.7759, Z -3.0000, A 0.000, B 0.000, C 0.000 }
gfCNCPoint2[6743] = {X 444.3934, Y 22.7960, Z -3.0000, A 0.000, B 0.000, C 0.000 }
gfCNCPoint2[6744] = {X 445.9282, Y 22.7960, Z -3.0000, A 0.000, B 0.000, C 0.000 }
gfCNCPoint2[6745] = {X 449.9130, Y 22.4474, Z -3.0000, A 0.000, B 0.000, C 0.000 }
gfCNCPoint2[6746] = {X 441.9435, Y 22.5274, Z -3.0000, A 0.000, B 0.000, C 0.000 }
gfCNCPoint2[6747] = {X 445.9282, Y 22.8760, Z -3.0000, A 0.000, B 0.000, C 0.000 }
gfCNCPoint2[6748] = {X 450.4384, Y 22.8760, Z -3.0000, A 0.000, B 0.000, C 0.000 }
gfCNCPoint2[6749] = {X 450.4384, Y 19.4614, Z -3.0000, A 0.000, B 0.000, C 0.000 }
gfCNCPoint2[6750] = {X 444.0376, Y 19.4611, Z -3.0000, A 0.000, B 0.000, C 0.000 }
gfCNCPoint2[6751] = {X 443.3456, Y 19.4773, Z -3.0000, A 0.000, B 0.000, C 0.000 }
gfCNCPoint2[6752] = {X 442.3416, Y 19.5695, Z -3.0000, A 0.000, B 0.000, C 0.000 }
gfCNCPoint2[6753] = {X 441.3650, Y 19.8202, Z -3.0000, A 0.000, B 0.000, C 0.000 }
gfCNCPoint2[6754] = {X 441.1557, Y 19.9526, Z -3.0000, A 0.000, B 0.000, C 0.000 }
gfCNCPoint2[6755] = {X 441.0281, Y 20.1650, Z -3.0000, A 0.000, B 0.000, C 0.000 }
gfCNCPoint2[6756] = {X 440.8586, Y 20.9684, Z -3.0000, A 0.000, B 0.000, C 0.000 }
gfCNCPoint2[6757] = {X 440.8519, Y 21.7895, Z -3.0000, A 0.000, B 0.000, C 0.000 }
gfCNCPoint2[6758] = {X 441.0085, Y 22.5955, Z -3.0000, A 0.000, B 0.000, C 0.000 }
gfCNCPoint2[6759] = {X 441.3539, Y 22.7076, Z -3.0000, A 0.000, B 0.000, C 0.000 }
gfCNCPoint2[6760] = {X 441.7121, Y 22.7675, Z -3.0000, A 0.000, B 0.000, C 0.000 }
gfCNCPoint2[6761] = {X 443.0516, Y 22.8559, Z -3.0000, A 0.000, B 0.000, C 0.000 }
gfCNCPoint2[6762] = {X 444.3938, Y 22.8760, Z -3.0000, A 0.000, B 0.000, C 0.000 }
gfCNCPoint2[6763] = {X 445.9282, Y 22.8760, Z -3.0000, A 0.000, B 0.000, C 0.000 }
gfCNCPoint2[6764] = {X 449.9130, Y 22.5274, Z -3.0000, A 0.000, B 0.000, C 0.000 }
gfCNCPoint2[6765] = {X 441.9435, Y 22.6074, Z -3.0000, A 0.000, B 0.000, C 0.000 }
gfCNCPoint2[6766] = {X 445.9282, Y 22.9560, Z -3.0000, A 0.000, B 0.000, C 0.000 }
gfCNCPoint2[6767] = {X 450.5184, Y 22.9560, Z -3.0000, A 0.000, B 0.000, C 0.000 }
gfCNCPoint2[6768] = {X 450.5194, Y 19.3814, Z -3.0000, A 0.000, B 0.000, C 0.000 }
gfCNCPoint2[6769] = {X 444.0367, Y 19.3811, Z -3.0000, A 0.000, B 0.000, C 0.000 }
gfCNCPoint2[6770] = {X 443.3442, Y 19.3973, Z -3.0000, A 0.000, B 0.000, C 0.000 }
gfCNCPoint2[6771] = {X 442.3277, Y 19.4907, Z -3.0000, A 0.000, B 0.000, C 0.000 }
gfCNCPoint2[6772] = {X 441.3390, Y 19.7445, Z -3.0000, A 0.000, B 0.000, C 0.000 }
gfCNCPoint2[6773] = {X 441.0984, Y 19.8967, Z -3.0000, A 0.000, B 0.000, C 0.000 }
gfCNCPoint2[6774] = {X 440.9519, Y 20.1407, Z -3.0000, A 0.000, B 0.000, C 0.000 }
gfCNCPoint2[6775] = {X 440.7777, Y 20.9724, Z -3.0000, A 0.000, B 0.000, C 0.000 }
gfCNCPoint2[6776] = {X 440.7747, Y 21.8220, Z -3.0000, A 0.000, B 0.000, C 0.000 }
gfCNCPoint2[6777] = {X 440.9429, Y 22.6549, Z -3.0000, A 0.000, B 0.000, C 0.000 }
gfCNCPoint2[6778] = {X 441.3164, Y 22.7807, Z -3.0000, A 0.000, B 0.000, C 0.000 }
gfCNCPoint2[6779] = {X 441.7048, Y 22.8471, Z -3.0000, A 0.000, B 0.000, C 0.000 }
gfCNCPoint2[6780] = {X 443.0482, Y 22.9358, Z -3.0000, A 0.000, B 0.000, C 0.000 }
gfCNCPoint2[6781] = {X 444.3942, Y 22.9560, Z -3.0000, A 0.000, B 0.000, C 0.000 }
gfCNCPoint2[6782] = {X 445.9282, Y 22.9560, Z -3.0000, A 0.000, B 0.000, C 0.000 }
gfCNCPoint2[6783] = {X 449.9130, Y 22.6074, Z -3.0000, A 0.000, B 0.000, C 0.000 }
gfCNCPoint2[6784] = {X 449.9130, Y 22.6074, Z 0.0000, A 0.000, B 0.000, C 0.000 }
gfCNCPoint2[6785] = {X 449.9130, Y 22.6074, Z 11.0000, A 0.000, B 0.000, C 0.000 }
gfCNCPoint2[6786] = {X 507.6818, Y 107.6950, Z 11.0000, A 0.000, B 0.000, C 0.000 }
gfCNCPoint2[6787] = {X 507.6818, Y 107.6950, Z 0.0000, A 0.000, B 0.000, C 0.000 }
gfCNCPoint2[6788] = {X 507.6818, Y 107.6950, Z -3.0000, A 0.000, B 0.000, C 0.000 }
gfCNCPoint2[6789] = {X 507.6818, Y 71.2950, Z -3.0000, A 0.000, B 0.000, C 0.000 }
gfCNCPoint2[6790] = {X 509.5500, Y 71.2950, Z -3.0000, A 0.000, B 0.000, C 0.000 }
gfCNCPoint2[6791] = {X 509.0278, Y 71.0691, Z -3.0000, A 0.000, B 0.000, C 0.000 }
gfCNCPoint2[6792] = {X 508.5105, Y 70.8320, Z -3.0000, A 0.000, B 0.000, C 0.000 }
gfCNCPoint2[6793] = {X 507.1680, Y 71.0984, Z -3.0000, A 0.000, B 0.000, C 0.000 }
gfCNCPoint2[6794] = {X 505.8135, Y 71.2950, Z -3.0000, A 0.000, B 0.000, C 0.000 }
gfCNCPoint2[6795] = {X 507.6818, Y 71.2950, Z -3.0000, A 0.000, B 0.000, C 0.000 }
gfCNCPoint2[6796] = {X 507.6818, Y 73.6950, Z -3.0000, A 0.000, B 0.000, C 0.000 }
gfCNCPoint2[6797] = {X 551.2533, Y 73.6950, Z -3.0000, A 0.000, B 0.000, C 0.000 }
gfCNCPoint2[6798] = {X 549.1234, Y 72.7704, Z -3.0000, A 0.000, B 0.000, C 0.000 }
gfCNCPoint2[6799] = {X 547.0693, Y 71.6880, Z -3.0000, A 0.000, B 0.000, C 0.000 }
gfCNCPoint2[6800] = {X 545.1026, Y 70.4540, Z -3.0000, A 0.000, B 0.000, C 0.000 }
gfCNCPoint2[6801] = {X 543.2344, Y 69.0753, Z -3.0000, A 0.000, B 0.000, C 0.000 }
gfCNCPoint2[6802] = {X 529.7638, Y 69.0756, Z -3.0000, A 0.000, B 0.000, C 0.000 }
gfCNCPoint2[6803] = {X 527.5499, Y 69.8794, Z -3.0000, A 0.000, B 0.000, C 0.000 }
gfCNCPoint2[6804] = {X 525.2685, Y 70.4646, Z -3.0000, A 0.000, B 0.000, C 0.000 }
gfCNCPoint2[6805] = {X 522.9410, Y 70.8256, Z -3.0000, A 0.000, B 0.000, C 0.000 }
gfCNCPoint2[6806] = {X 520.5895, Y 70.9589, Z -3.0000, A 0.000, B 0.000, C 0.000 }
gfCNCPoint2[6807] = {X 519.7998, Y 70.9591, Z -3.0000, A 0.000, B 0.000, C 0.000 }
gfCNCPoint2[6808] = {X 517.4110, Y 70.8403, Z -3.0000, A 0.000, B 0.000, C 0.000 }
gfCNCPoint2[6809] = {X 515.0458, Y 70.4852, Z -3.0000, A 0.000, B 0.000, C 0.000 }
gfCNCPoint2[6810] = {X 512.7275, Y 69.8972, Z -3.0000, A 0.000, B 0.000, C 0.000 }
gfCNCPoint2[6811] = {X 510.4790, Y 69.0820, Z -3.0000, A 0.000, B 0.000, C 0.000 }
gfCNCPoint2[6812] = {X 509.6265, Y 68.7046, Z -3.0000, A 0.000, B 0.000, C 0.000 }
gfCNCPoint2[6813] = {X 508.7892, Y 68.2944, Z -3.0000, A 0.000, B 0.000, C 0.000 }
gfCNCPoint2[6814] = {X 507.1704, Y 68.6592, Z -3.0000, A 0.000, B 0.000, C 0.000 }
gfCNCPoint2[6815] = {X 505.5302, Y 68.9117, Z -3.0000, A 0.000, B 0.000, C 0.000 }
gfCNCPoint2[6816] = {X 504.1119, Y 69.0379, Z -3.0000, A 0.000, B 0.000, C 0.000 }
gfCNCPoint2[6817] = {X 502.6885, Y 69.0800, Z -3.0000, A 0.000, B 0.000, C 0.000 }
gfCNCPoint2[6818] = {X 502.0391, Y 69.0800, Z -3.0000, A 0.000, B 0.000, C 0.000 }
gfCNCPoint2[6819] = {X 501.1773, Y 71.1326, Z -3.0000, A 0.000, B 0.000, C 0.000 }
gfCNCPoint2[6820] = {X 500.1599, Y 73.1128, Z -3.0000, A 0.000, B 0.000, C 0.000 }
gfCNCPoint2[6821] = {X 500.1599, Y 73.6950, Z -3.0000, A 0.000, B 0.000, C 0.000 }
gfCNCPoint2[6822] = {X 507.6818, Y 73.6950, Z -3.0000, A 0.000, B 0.000, C 0.000 }
gfCNCPoint2[6823] = {X 507.6818, Y 76.0950, Z -3.0000, A 0.000, B 0.000, C 0.000 }
gfCNCPoint2[6824] = {X 576.0965, Y 76.0950, Z -3.0000, A 0.000, B 0.000, C 0.000 }
gfCNCPoint2[6825] = {X 576.0965, Y 72.8901, Z -3.0000, A 0.000, B 0.000, C 0.000 }
gfCNCPoint2[6826] = {X 575.7178, Y 72.8147, Z -3.0000, A 0.000, B 0.000, C 0.000 }
gfCNCPoint2[6827] = {X 575.3401, Y 72.7341, Z -3.0000, A 0.000, B 0.000, C 0.000 }
gfCNCPoint2[6828] = {X 573.3201, Y 73.1034, Z -3.0000, A 0.000, B 0.000, C 0.000 }
gfCNCPoint2[6829] = {X 571.2786, Y 73.3258, Z -3.0000, A 0.000, B 0.000, C 0.000 }
gfCNCPoint2[6830] = {X 569.2264, Y 73.4000, Z -3.0000, A 0.000, B 0.000, C 0.000 }
gfCNCPoint2[6831] = {X 562.4443, Y 73.4000, Z -3.0000, A 0.000, B 0.000, C 0.000 }
gfCNCPoint2[6832] = {X 560.3341, Y 73.3215, Z -3.0000, A 0.000, B 0.000, C 0.000 }
gfCNCPoint2[6833] = {X 558.2356, Y 73.0864, Z -3.0000, A 0.000, B 0.000, C 0.000 }
gfCNCPoint2[6834] = {X 556.1603, Y 72.6961, Z -3.0000, A 0.000, B 0.000, C 0.000 }
gfCNCPoint2[6835] = {X 554.1198, Y 72.1526, Z -3.0000, A 0.000, B 0.000, C 0.000 }
gfCNCPoint2[6836] = {X 552.1253, Y 71.4590, Z -3.0000, A 0.000, B 0.000, C 0.000 }
gfCNCPoint2[6837] = {X 549.9759, Y 70.5166, Z -3.0000, A 0.000, B 0.000, C 0.000 }
gfCNCPoint2[6838] = {X 547.9116, Y 69.4000, Z -3.0000, A 0.000, B 0.000, C 0.000 }
gfCNCPoint2[6839] = {X 545.9466, Y 68.1168, Z -3.0000, A 0.000, B 0.000, C 0.000 }
gfCNCPoint2[6840] = {X 544.0942, Y 66.6756, Z -3.0000, A 0.000, B 0.000, C 0.000 }
gfCNCPoint2[6841] = {X 543.8497, Y 66.6768, Z -3.0000, A 0.000, B 0.000, C 0.000 }
gfCNCPoint2[6842] = {X 543.6053, Y 66.6753, Z -3.0000, A 0.000, B 0.000, C 0.000 }
gfCNCPoint2[6843] = {X 529.2681, Y 66.6756, Z -3.0000, A 0.000, B 0.000, C 0.000 }
gfCNCPoint2[6844] = {X 527.1777, Y 67.4795, Z -3.0000, A 0.000, B 0.000, C 0.000 }
gfCNCPoint2[6845] = {X 525.0160, Y 68.0651, Z -3.0000, A 0.000, B 0.000, C 0.000 }
gfCNCPoint2[6846] = {X 522.8057, Y 68.4262, Z -3.0000, A 0.000, B 0.000, C 0.000 }
gfCNCPoint2[6847] = {X 520.5701, Y 68.5590, Z -3.0000, A 0.000, B 0.000, C 0.000 }
gfCNCPoint2[6848] = {X 519.7998, Y 68.5591, Z -3.0000, A 0.000, B 0.000, C 0.000 }
gfCNCPoint2[6849] = {X 517.5593, Y 68.4430, Z -3.0000, A 0.000, B 0.000, C 0.000 }
gfCNCPoint2[6850] = {X 515.3429, Y 68.0961, Z -3.0000, A 0.000, B 0.000, C 0.000 }
gfCNCPoint2[6851] = {X 513.1742, Y 67.5219, Z -3.0000, A 0.000, B 0.000, C 0.000 }
gfCNCPoint2[6852] = {X 511.0764, Y 66.7267, Z -3.0000, A 0.000, B 0.000, C 0.000 }
gfCNCPoint2[6853] = {X 509.0720, Y 65.7189, Z -3.0000, A 0.000, B 0.000, C 0.000 }
gfCNCPoint2[6854] = {X 506.9797, Y 66.2511, Z -3.0000, A 0.000, B 0.000, C 0.000 }
gfCNCPoint2[6855] = {X 504.8448, Y 66.5725, Z -3.0000, A 0.000, B 0.000, C 0.000 }
gfCNCPoint2[6856] = {X 502.6885, Y 66.6800, Z -3.0000, A 0.000, B 0.000, C 0.000 }
gfCNCPoint2[6857] = {X 500.3217, Y 66.6800, Z -3.0000, A 0.000, B 0.000, C 0.000 }
gfCNCPoint2[6858] = {X 499.6230, Y 68.6757, Z -3.0000, A 0.000, B 0.000, C 0.000 }
gfCNCPoint2[6859] = {X 498.7672, Y 70.6093, Z -3.0000, A 0.000, B 0.000, C 0.000 }
gfCNCPoint2[6860] = {X 497.7599, Y 72.4684, Z -3.0000, A 0.000, B 0.000, C 0.000 }
gfCNCPoint2[6861] = {X 497.7599, Y 76.0950, Z -3.0000, A 0.000, B 0.000, C 0.000 }
gfCNCPoint2[6862] = {X 507.6818, Y 76.0950, Z -3.0000, A 0.000, B 0.000, C 0.000 }
gfCNCPoint2[6863] = {X 507.6818, Y 78.4950, Z -3.0000, A 0.000, B 0.000, C 0.000 }
gfCNCPoint2[6864] = {X 578.4965, Y 78.4950, Z -3.0000, A 0.000, B 0.000, C 0.000 }
gfCNCPoint2[6865] = {X 578.4965, Y 70.8313, Z -3.0000, A 0.000, B 0.000, C 0.000 }
gfCNCPoint2[6866] = {X 576.9097, Y 70.5998, Z -3.0000, A 0.000, B 0.000, C 0.000 }
gfCNCPoint2[6867] = {X 575.3401, Y 70.2710, Z -3.0000, A 0.000, B 0.000, C 0.000 }
gfCNCPoint2[6868] = {X 573.3236, Y 70.6751, Z -3.0000, A 0.000, B 0.000, C 0.000 }
gfCNCPoint2[6869] = {X 571.2815, Y 70.9187, Z -3.0000, A 0.000, B 0.000, C 0.000 }
gfCNCPoint2[6870] = {X 569.2264, Y 71.0000, Z -3.0000, A 0.000, B 0.000, C 0.000 }
gfCNCPoint2[6871] = {X 562.4443, Y 71.0000, Z -3.0000, A 0.000, B 0.000, C 0.000 }
gfCNCPoint2[6872] = {X 560.0511, Y 70.8896, Z -3.0000, A 0.000, B 0.000, C 0.000 }
gfCNCPoint2[6873] = {X 557.6783, Y 70.5594, Z -3.0000, A 0.000, B 0.000, C 0.000 }
gfCNCPoint2[6874] = {X 555.3459, Y 70.0123, Z -3.0000, A 0.000, B 0.000, C 0.000 }
gfCNCPoint2[6875] = {X 553.0738, Y 69.2527, Z -3.0000, A 0.000, B 0.000, C 0.000 }
gfCNCPoint2[6876] = {X 550.8813, Y 68.2872, Z -3.0000, A 0.000, B 0.000, C 0.000 }
gfCNCPoint2[6877] = {X 548.7869, Y 67.1241, Z -3.0000, A 0.000, B 0.000, C 0.000 }
gfCNCPoint2[6878] = {X 546.8084, Y 65.7731, Z -3.0000, A 0.000, B 0.000, C 0.000 }
gfCNCPoint2[6879] = {X 544.9628, Y 64.2457, Z -3.0000, A 0.000, B 0.000, C 0.000 }
gfCNCPoint2[6880] = {X 544.2917, Y 64.2722, Z -3.0000, A 0.000, B 0.000, C 0.000 }
gfCNCPoint2[6881] = {X 543.6202, Y 64.2753, Z -3.0000, A 0.000, B 0.000, C 0.000 }
gfCNCPoint2[6882] = {X 528.7429, Y 64.2756, Z -3.0000, A 0.000, B 0.000, C 0.000 }
gfCNCPoint2[6883] = {X 526.7864, Y 65.0787, Z -3.0000, A 0.000, B 0.000, C 0.000 }
gfCNCPoint2[6884] = {X 524.7542, Y 65.6645, Z -3.0000, A 0.000, B 0.000, C 0.000 }
gfCNCPoint2[6885] = {X 522.6704, Y 66.0260, Z -3.0000, A 0.000, B 0.000, C 0.000 }
gfCNCPoint2[6886] = {X 520.5597, Y 66.1590, Z -3.0000, A 0.000, B 0.000, C 0.000 }
gfCNCPoint2[6887] = {X 519.7998, Y 66.1591, Z -3.0000, A 0.000, B 0.000, C 0.000 }
gfCNCPoint2[6888] = {X 517.9641, Y 66.0715, Z -3.0000, A 0.000, B 0.000, C 0.000 }
gfCNCPoint2[6889] = {X 516.1450, Y 65.8096, Z -3.0000, A 0.000, B 0.000, C 0.000 }
gfCNCPoint2[6890] = {X 514.3592, Y 65.3756, Z -3.0000, A 0.000, B 0.000, C 0.000 }
gfCNCPoint2[6891] = {X 512.6228, Y 64.7735, Z -3.0000, A 0.000, B 0.000, C 0.000 }
gfCNCPoint2[6892] = {X 510.9516, Y 64.0089, Z -3.0000, A 0.000, B 0.000, C 0.000 }
gfCNCPoint2[6893] = {X 509.3609, Y 63.0886, Z -3.0000, A 0.000, B 0.000, C 0.000 }
gfCNCPoint2[6894] = {X 507.7389, Y 63.6068, Z -3.0000, A 0.000, B 0.000, C 0.000 }
gfCNCPoint2[6895] = {X 506.0774, Y 63.9798, Z -3.0000, A 0.000, B 0.000, C 0.000 }
gfCNCPoint2[6896] = {X 504.3896, Y 64.2048, Z -3.0000, A 0.000, B 0.000, C 0.000 }
gfCNCPoint2[6897] = {X 502.6885, Y 64.2800, Z -3.0000, A 0.000, B 0.000, C 0.000 }
gfCNCPoint2[6898] = {X 498.4791, Y 64.2800, Z -3.0000, A 0.000, B 0.000, C 0.000 }
gfCNCPoint2[6899] = {X 497.9415, Y 66.2506, Z -3.0000, A 0.000, B 0.000, C 0.000 }
gfCNCPoint2[6900] = {X 497.2389, Y 68.1686, Z -3.0000, A 0.000, B 0.000, C 0.000 }
gfCNCPoint2[6901] = {X 496.3763, Y 70.0201, Z -3.0000, A 0.000, B 0.000, C 0.000 }
gfCNCPoint2[6902] = {X 495.3598, Y 71.7919, Z -3.0000, A 0.000, B 0.000, C 0.000 }
gfCNCPoint2[6903] = {X 495.3599, Y 78.4950, Z -3.0000, A 0.000, B 0.000, C 0.000 }
gfCNCPoint2[6904] = {X 507.6818, Y 78.4950, Z -3.0000, A 0.000, B 0.000, C 0.000 }
gfCNCPoint2[6905] = {X 507.6818, Y 80.8950, Z -3.0000, A 0.000, B 0.000, C 0.000 }
gfCNCPoint2[6906] = {X 580.8965, Y 80.8950, Z -3.0000, A 0.000, B 0.000, C 0.000 }
gfCNCPoint2[6907] = {X 580.8965, Y 68.5934, Z -3.0000, A 0.000, B 0.000, C 0.000 }
gfCNCPoint2[6908] = {X 579.0252, Y 68.4747, Z -3.0000, A 0.000, B 0.000, C 0.000 }
gfCNCPoint2[6909] = {X 577.1691, Y 68.2078, Z -3.0000, A 0.000, B 0.000, C 0.000 }
gfCNCPoint2[6910] = {X 575.3401, Y 67.7943, Z -3.0000, A 0.000, B 0.000, C 0.000 }
gfCNCPoint2[6911] = {X 573.3283, Y 68.2408, Z -3.0000, A 0.000, B 0.000, C 0.000 }
gfCNCPoint2[6912] = {X 571.2852, Y 68.5100, Z -3.0000, A 0.000, B 0.000, C 0.000 }
gfCNCPoint2[6913] = {X 569.2264, Y 68.6000, Z -3.0000, A 0.000, B 0.000, C 0.000 }
gfCNCPoint2[6914] = {X 562.4443, Y 68.6000, Z -3.0000, A 0.000, B 0.000, C 0.000 }
gfCNCPoint2[6915] = {X 560.1442, Y 68.4876, Z -3.0000, A 0.000, B 0.000, C 0.000 }
gfCNCPoint2[6916] = {X 557.8660, Y 68.1517, Z -3.0000, A 0.000, B 0.000, C 0.000 }
gfCNCPoint2[6917] = {X 555.6315, Y 67.5952, Z -3.0000, A 0.000, B 0.000, C 0.000 }
gfCNCPoint2[6918] = {X 553.4617, Y 66.8237, Z -3.0000, A 0.000, B 0.000, C 0.000 }
gfCNCPoint2[6919] = {X 551.3775, Y 65.8443, Z -3.0000, A 0.000, B 0.000, C 0.000 }
gfCNCPoint2[6920] = {X 549.3987, Y 64.6665, Z -3.0000, A 0.000, B 0.000, C 0.000 }
gfCNCPoint2[6921] = {X 547.5441, Y 63.3015, Z -3.0000, A 0.000, B 0.000, C 0.000 }
gfCNCPoint2[6922] = {X 545.8314, Y 61.7622, Z -3.0000, A 0.000, B 0.000, C 0.000 }
gfCNCPoint2[6923] = {X 544.7355, Y 61.8545, Z -3.0000, A 0.000, B 0.000, C 0.000 }
gfCNCPoint2[6924] = {X 543.6360, Y 61.8753, Z -3.0000, A 0.000, B 0.000, C 0.000 }
gfCNCPoint2[6925] = {X 528.1825, Y 61.8757, Z -3.0000, A 0.000, B 0.000, C 0.000 }
gfCNCPoint2[6926] = {X 526.3695, Y 62.6777, Z -3.0000, A 0.000, B 0.000, C 0.000 }
gfCNCPoint2[6927] = {X 524.4757, Y 63.2637, Z -3.0000, A 0.000, B 0.000, C 0.000 }
gfCNCPoint2[6928] = {X 522.5266, Y 63.6258, Z -3.0000, A 0.000, B 0.000, C 0.000 }
gfCNCPoint2[6929] = {X 520.5487, Y 63.7590, Z -3.0000, A 0.000, B 0.000, C 0.000 }
gfCNCPoint2[6930] = {X 519.7998, Y 63.7591, Z -3.0000, A 0.000, B 0.000, C 0.000 }
gfCNCPoint2[6931] = {X 517.9902, Y 63.6618, Z -3.0000, A 0.000, B 0.000, C 0.000 }
gfCNCPoint2[6932] = {X 516.2015, Y 63.3711, Z -3.0000, A 0.000, B 0.000, C 0.000 }
gfCNCPoint2[6933] = {X 514.4543, Y 62.8904, Z -3.0000, A 0.000, B 0.000, C 0.000 }
gfCNCPoint2[6934] = {X 512.7687, Y 62.2251, Z -3.0000, A 0.000, B 0.000, C 0.000 }
gfCNCPoint2[6935] = {X 511.1641, Y 61.3829, Z -3.0000, A 0.000, B 0.000, C 0.000 }
gfCNCPoint2[6936] = {X 509.6590, Y 60.3735, Z -3.0000, A 0.000, B 0.000, C 0.000 }
gfCNCPoint2[6937] = {X 507.9866, Y 61.0270, Z -3.0000, A 0.000, B 0.000, C 0.000 }
gfCNCPoint2[6938] = {X 506.2542, Y 61.4991, Z -3.0000, A 0.000, B 0.000, C 0.000 }
gfCNCPoint2[6939] = {X 504.4815, Y 61.7845, Z -3.0000, A 0.000, B 0.000, C 0.000 }
gfCNCPoint2[6940] = {X 502.6885, Y 61.8800, Z -3.0000, A 0.000, B 0.000, C 0.000 }
gfCNCPoint2[6941] = {X 496.4789, Y 61.8800, Z -3.0000, A 0.000, B 0.000, C 0.000 }
gfCNCPoint2[6942] = {X 496.1192, Y 63.8334, Z -3.0000, A 0.000, B 0.000, C 0.000 }
gfCNCPoint2[6943] = {X 495.5822, Y 65.7456, Z -3.0000, A 0.000, B 0.000, C 0.000 }
gfCNCPoint2[6944] = {X 494.8724, Y 67.6007, Z -3.0000, A 0.000, B 0.000, C 0.000 }
gfCNCPoint2[6945] = {X 493.9958, Y 69.3830, Z -3.0000, A 0.000, B 0.000, C 0.000 }
gfCNCPoint2[6946] = {X 492.9598, Y 71.0777, Z -3.0000, A 0.000, B 0.000, C 0.000 }
gfCNCPoint2[6947] = {X 492.9600, Y 80.8950, Z -3.0000, A 0.000, B 0.000, C 0.000 }
gfCNCPoint2[6948] = {X 507.6818, Y 80.8950, Z -3.0000, A 0.000, B 0.000, C 0.000 }
gfCNCPoint2[6949] = {X 507.6818, Y 83.2950, Z -3.0000, A 0.000, B 0.000, C 0.000 }
gfCNCPoint2[6950] = {X 583.2965, Y 83.2950, Z -3.0000, A 0.000, B 0.000, C 0.000 }
gfCNCPoint2[6951] = {X 583.2965, Y 66.1198, Z -3.0000, A 0.000, B 0.000, C 0.000 }
gfCNCPoint2[6952] = {X 581.2872, Y 66.1993, Z -3.0000, A 0.000, B 0.000, C 0.000 }
gfCNCPoint2[6953] = {X 579.2793, Y 66.0882, Z -3.0000, A 0.000, B 0.000, C 0.000 }
gfCNCPoint2[6954] = {X 577.2910, Y 65.7873, Z -3.0000, A 0.000, B 0.000, C 0.000 }
gfCNCPoint2[6955] = {X 575.3401, Y 65.2993, Z -3.0000, A 0.000, B 0.000, C 0.000 }
gfCNCPoint2[6956] = {X 573.3348, Y 65.7981, Z -3.0000, A 0.000, B 0.000, C 0.000 }
gfCNCPoint2[6957] = {X 571.2904, Y 66.0993, Z -3.0000, A 0.000, B 0.000, C 0.000 }
gfCNCPoint2[6958] = {X 569.2264, Y 66.2000, Z -3.0000, A 0.000, B 0.000, C 0.000 }
gfCNCPoint2[6959] = {X 562.4443, Y 66.2000, Z -3.0000, A 0.000, B 0.000, C 0.000 }
gfCNCPoint2[6960] = {X 560.2302, Y 66.0841, Z -3.0000, A 0.000, B 0.000, C 0.000 }
gfCNCPoint2[6961] = {X 558.0404, Y 65.7375, Z -3.0000, A 0.000, B 0.000, C 0.000 }
gfCNCPoint2[6962] = {X 555.8987, Y 65.1642, Z -3.0000, A 0.000, B 0.000, C 0.000 }
gfCNCPoint2[6963] = {X 553.8286, Y 64.3703, Z -3.0000, A 0.000, B 0.000, C 0.000 }
gfCNCPoint2[6964] = {X 551.8527, Y 63.3646, Z -3.0000, A 0.000, B 0.000, C 0.000 }
gfCNCPoint2[6965] = {X 549.9926, Y 62.1580, Z -3.0000, A 0.000, B 0.000, C 0.000 }
gfCNCPoint2[6966] = {X 548.2688, Y 60.7637, Z -3.0000, A 0.000, B 0.000, C 0.000 }
gfCNCPoint2[6967] = {X 546.7000, Y 59.1971, Z -3.0000, A 0.000, B 0.000, C 0.000 }
gfCNCPoint2[6968] = {X 545.1839, Y 59.4168, Z -3.0000, A 0.000, B 0.000, C 0.000 }
gfCNCPoint2[6969] = {X 543.6530, Y 59.4753, Z -3.0000, A 0.000, B 0.000, C 0.000 }
gfCNCPoint2[6970] = {X 527.5784, Y 59.4757, Z -3.0000, A 0.000, B 0.000, C 0.000 }
gfCNCPoint2[6971] = {X 525.9212, Y 60.2763, Z -3.0000, A 0.000, B 0.000, C 0.000 }
gfCNCPoint2[6972] = {X 524.1767, Y 60.8626, Z -3.0000, A 0.000, B 0.000, C 0.000 }
gfCNCPoint2[6973] = {X 522.3724, Y 61.2255, Z -3.0000, A 0.000, B 0.000, C 0.000 }
gfCNCPoint2[6974] = {X 520.5368, Y 61.3590, Z -3.0000, A 0.000, B 0.000, C 0.000 }
gfCNCPoint2[6975] = {X 519.7998, Y 61.3591, Z -3.0000, A 0.000, B 0.000, C 0.000 }
gfCNCPoint2[6976] = {X 518.0043, Y 61.2474, Z -3.0000, A 0.000, B 0.000, C 0.000 }
gfCNCPoint2[6977] = {X 516.2365, Y 60.9138, Z -3.0000, A 0.000, B 0.000, C 0.000 }
gfCNCPoint2[6978] = {X 514.5237, Y 60.3637, Z -3.0000, A 0.000, B 0.000, C 0.000 }
gfCNCPoint2[6979] = {X 512.8923, Y 59.6054, Z -3.0000, A 0.000, B 0.000, C 0.000 }
gfCNCPoint2[6980] = {X 511.3676, Y 58.6507, Z -3.0000, A 0.000, B 0.000, C 0.000 }
gfCNCPoint2[6981] = {X 509.9730, Y 57.5142, Z -3.0000, A 0.000, B 0.000, C 0.000 }
gfCNCPoint2[6982] = {X 508.6156, Y 58.2113, Z -3.0000, A 0.000, B 0.000, C 0.000 }
gfCNCPoint2[6983] = {X 507.1924, Y 58.7617, Z -3.0000, A 0.000, B 0.000, C 0.000 }
gfCNCPoint2[6984] = {X 505.7192, Y 59.1593, Z -3.0000, A 0.000, B 0.000, C 0.000 }
gfCNCPoint2[6985] = {X 504.2123, Y 59.3996, Z -3.0000, A 0.000, B 0.000, C 0.000 }
gfCNCPoint2[6986] = {X 502.6885, Y 59.4800, Z -3.0000, A 0.000, B 0.000, C 0.000 }
gfCNCPoint2[6987] = {X 496.2450, Y 59.4800, Z -3.0000, A 0.000, B 0.000, C 0.000 }
gfCNCPoint2[6988] = {X 495.2580, Y 59.4463, Z -3.0000, A 0.000, B 0.000, C 0.000 }
gfCNCPoint2[6989] = {X 494.2756, Y 59.3454, Z -3.0000, A 0.000, B 0.000, C 0.000 }
gfCNCPoint2[6990] = {X 494.1342, Y 61.3007, Z -3.0000, A 0.000, B 0.000, C 0.000 }
gfCNCPoint2[6991] = {X 493.7950, Y 63.2314, Z -3.0000, A 0.000, B 0.000, C 0.000 }
gfCNCPoint2[6992] = {X 493.2614, Y 65.1178, Z -3.0000, A 0.000, B 0.000, C 0.000 }
gfCNCPoint2[6993] = {X 492.5391, Y 66.9402, Z -3.0000, A 0.000, B 0.000, C 0.000 }
gfCNCPoint2[6994] = {X 491.6355, Y 68.6798, Z -3.0000, A 0.000, B 0.000, C 0.000 }
gfCNCPoint2[6995] = {X 490.5598, Y 70.3187, Z -3.0000, A 0.000, B 0.000, C 0.000 }
gfCNCPoint2[6996] = {X 490.5600, Y 83.2950, Z -3.0000, A 0.000, B 0.000, C 0.000 }
gfCNCPoint2[6997] = {X 507.6818, Y 83.2950, Z -3.0000, A 0.000, B 0.000, C 0.000 }
gfCNCPoint2[6998] = {X 507.6818, Y 85.6950, Z -3.0000, A 0.000, B 0.000, C 0.000 }
gfCNCPoint2[6999] = {X 585.6965, Y 85.6950, Z -3.0000, A 0.000, B 0.000, C 0.000 }
gfCNCPoint2[7000] = {X 585.6965, Y 63.3150, Z -3.0000, A 0.000, B 0.000, C 0.000 }
gfCNCPoint2[7001] = {X 584.3995, Y 63.5678, Z -3.0000, A 0.000, B 0.000, C 0.000 }
gfCNCPoint2[7002] = {X 583.0879, Y 63.7288, Z -3.0000, A 0.000, B 0.000, C 0.000 }
gfCNCPoint2[7003] = {X 581.1242, Y 63.7971, Z -3.0000, A 0.000, B 0.000, C 0.000 }
gfCNCPoint2[7004] = {X 579.1641, Y 63.6600, Z -3.0000, A 0.000, B 0.000, C 0.000 }
gfCNCPoint2[7005] = {X 577.2291, Y 63.3191, Z -3.0000, A 0.000, B 0.000, C 0.000 }
gfCNCPoint2[7006] = {X 575.3401, Y 62.7781, Z -3.0000, A 0.000, B 0.000, C 0.000 }
gfCNCPoint2[7007] = {X 573.3441, Y 63.3435, Z -3.0000, A 0.000, B 0.000, C 0.000 }
gfCNCPoint2[7008] = {X 571.2979, Y 63.6855, Z -3.0000, A 0.000, B 0.000, C 0.000 }
gfCNCPoint2[7009] = {X 569.2264, Y 63.8000, Z -3.0000, A 0.000, B 0.000, C 0.000 }
gfCNCPoint2[7010] = {X 562.4443, Y 63.8000, Z -3.0000, A 0.000, B 0.000, C 0.000 }
gfCNCPoint2[7011] = {X 560.5407, Y 63.7034, Z -3.0000, A 0.000, B 0.000, C 0.000 }
gfCNCPoint2[7012] = {X 558.6567, Y 63.4145, Z -3.0000, A 0.000, B 0.000, C 0.000 }
gfCNCPoint2[7013] = {X 556.8116, Y 62.9363, Z -3.0000, A 0.000, B 0.000, C 0.000 }
gfCNCPoint2[7014] = {X 555.0244, Y 62.2738, Z -3.0000, A 0.000, B 0.000, C 0.000 }
gfCNCPoint2[7015] = {X 553.3134, Y 61.4337, Z -3.0000, A 0.000, B 0.000, C 0.000 }
gfCNCPoint2[7016] = {X 551.6964, Y 60.4247, Z -3.0000, A 0.000, B 0.000, C 0.000 }
gfCNCPoint2[7017] = {X 550.1898, Y 59.2572, Z -3.0000, A 0.000, B 0.000, C 0.000 }
gfCNCPoint2[7018] = {X 548.8091, Y 57.9430, Z -3.0000, A 0.000, B 0.000, C 0.000 }
gfCNCPoint2[7019] = {X 547.5687, Y 56.4959, Z -3.0000, A 0.000, B 0.000, C 0.000 }
gfCNCPoint2[7020] = {X 546.2933, Y 56.8307, Z -3.0000, A 0.000, B 0.000, C 0.000 }
gfCNCPoint2[7021] = {X 544.9891, Y 57.0246, Z -3.0000, A 0.000, B 0.000, C 0.000 }
gfCNCPoint2[7022] = {X 543.6715, Y 57.0753, Z -3.0000, A 0.000, B 0.000, C 0.000 }
gfCNCPoint2[7023] = {X 526.9187, Y 57.0757, Z -3.0000, A 0.000, B 0.000, C 0.000 }
gfCNCPoint2[7024] = {X 525.4307, Y 57.8754, Z -3.0000, A 0.000, B 0.000, C 0.000 }
gfCNCPoint2[7025] = {X 523.8469, Y 58.4627, Z -3.0000, A 0.000, B 0.000, C 0.000 }
gfCNCPoint2[7026] = {X 522.1972, Y 58.8262, Z -3.0000, A 0.000, B 0.000, C 0.000 }
gfCNCPoint2[7027] = {X 520.5132, Y 58.9591, Z -3.0000, A 0.000, B 0.000, C 0.000 }
gfCNCPoint2[7028] = {X 519.7998, Y 58.9591, Z -3.0000, A 0.000, B 0.000, C 0.000 }
gfCNCPoint2[7029] = {X 518.2467, Y 58.8589, Z -3.0000, A 0.000, B 0.000, C 0.000 }
gfCNCPoint2[7030] = {X 516.7195, Y 58.5598, Z -3.0000, A 0.000, B 0.000, C 0.000 }
gfCNCPoint2[7031] = {X 515.2433, Y 58.0668, Z -3.0000, A 0.000, B 0.000, C 0.000 }
gfCNCPoint2[7032] = {X 513.8428, Y 57.3882, Z -3.0000, A 0.000, B 0.000, C 0.000 }
gfCNCPoint2[7033] = {X 512.5411, Y 56.5351, Z -3.0000, A 0.000, B 0.000, C 0.000 }
gfCNCPoint2[7034] = {X 511.3600, Y 55.5218, Z -3.0000, A 0.000, B 0.000, C 0.000 }
gfCNCPoint2[7035] = {X 510.3189, Y 54.3650, Z -3.0000, A 0.000, B 0.000, C 0.000 }
gfCNCPoint2[7036] = {X 508.9711, Y 55.3177, Z -3.0000, A 0.000, B 0.000, C 0.000 }
gfCNCPoint2[7037] = {X 507.5060, Y 56.0778, Z -3.0000, A 0.000, B 0.000, C 0.000 }
gfCNCPoint2[7038] = {X 505.9510, Y 56.6311, Z -3.0000, A 0.000, B 0.000, C 0.000 }
gfCNCPoint2[7039] = {X 504.3351, Y 56.9672, Z -3.0000, A 0.000, B 0.000, C 0.000 }
gfCNCPoint2[7040] = {X 502.6885, Y 57.0800, Z -3.0000, A 0.000, B 0.000, C 0.000 }
gfCNCPoint2[7041] = {X 496.2450, Y 57.0800, Z -3.0000, A 0.000, B 0.000, C 0.000 }
gfCNCPoint2[7042] = {X 495.4216, Y 57.0519, Z -3.0000, A 0.000, B 0.000, C 0.000 }
gfCNCPoint2[7043] = {X 494.6020, Y 56.9677, Z -3.0000, A 0.000, B 0.000, C 0.000 }
gfCNCPoint2[7044] = {X 493.1719, Y 56.6826, Z -3.0000, A 0.000, B 0.000, C 0.000 }
gfCNCPoint2[7045] = {X 491.7866, Y 56.2272, Z -3.0000, A 0.000, B 0.000, C 0.000 }
gfCNCPoint2[7046] = {X 491.8566, Y 57.1124, Z -3.0000, A 0.000, B 0.000, C 0.000 }
gfCNCPoint2[7047] = {X 491.8800, Y 58.0000, Z -3.0000, A 0.000, B 0.000, C 0.000 }
gfCNCPoint2[7048] = {X 491.8794, Y 59.0735, Z -3.0000, A 0.000, B 0.000, C 0.000 }
gfCNCPoint2[7049] = {X 491.8782, Y 59.1839, Z -3.0000, A 0.000, B 0.000, C 0.000 }
gfCNCPoint2[7050] = {X 491.8762, Y 59.2942, Z -3.0000, A 0.000, B 0.000, C 0.000 }
gfCNCPoint2[7051] = {X 491.7363, Y 61.1319, Z -3.0000, A 0.000, B 0.000, C 0.000 }
gfCNCPoint2[7052] = {X 491.3969, Y 62.9434, Z -3.0000, A 0.000, B 0.000, C 0.000 }
gfCNCPoint2[7053] = {X 490.8621, Y 64.7071, Z -3.0000, A 0.000, B 0.000, C 0.000 }
gfCNCPoint2[7054] = {X 490.1382, Y 66.4019, Z -3.0000, A 0.000, B 0.000, C 0.000 }
gfCNCPoint2[7055] = {X 489.2339, Y 68.0078, Z -3.0000, A 0.000, B 0.000, C 0.000 }
gfCNCPoint2[7056] = {X 488.1598, Y 69.5054, Z -3.0000, A 0.000, B 0.000, C 0.000 }
gfCNCPoint2[7057] = {X 488.1600, Y 85.6950, Z -3.0000, A 0.000, B 0.000, C 0.000 }
gfCNCPoint2[7058] = {X 507.6818, Y 85.6950, Z -3.0000, A 0.000, B 0.000, C 0.000 }
gfCNCPoint2[7059] = {X 507.6818, Y 88.0950, Z -3.0000, A 0.000, B 0.000, C 0.000 }
gfCNCPoint2[7060] = {X 588.0965, Y 88.0950, Z -3.0000, A 0.000, B 0.000, C 0.000 }
gfCNCPoint2[7061] = {X 588.0965, Y 60.4644, Z -3.0000, A 0.000, B 0.000, C 0.000 }
gfCNCPoint2[7062] = {X 587.7998, Y 60.3564, Z -3.0000, A 0.000, B 0.000, C 0.000 }
gfCNCPoint2[7063] = {X 587.5052, Y 60.2427, Z -3.0000, A 0.000, B 0.000, C 0.000 }
gfCNCPoint2[7064] = {X 586.3438, Y 60.6540, Z -3.0000, A 0.000, B 0.000, C 0.000 }
gfCNCPoint2[7065] = {X 585.1549, Y 60.9769, Z -3.0000, A 0.000, B 0.000, C 0.000 }
gfCNCPoint2[7066] = {X 583.5152, Y 61.2699, Z -3.0000, A 0.000, B 0.000, C 0.000 }
gfCNCPoint2[7067] = {X 581.8543, Y 61.3951, Z -3.0000, A 0.000, B 0.000, C 0.000 }
gfCNCPoint2[7068] = {X 580.1892, Y 61.3512, Z -3.0000, A 0.000, B 0.000, C 0.000 }
gfCNCPoint2[7069] = {X 578.5372, Y 61.1386, Z -3.0000, A 0.000, B 0.000, C 0.000 }
gfCNCPoint2[7070] = {X 576.9153, Y 60.7595, Z -3.0000, A 0.000, B 0.000, C 0.000 }
gfCNCPoint2[7071] = {X 575.3401, Y 60.2178, Z -3.0000, A 0.000, B 0.000, C 0.000 }
gfCNCPoint2[7072] = {X 573.8611, Y 60.7315, Z -3.0000, A 0.000, B 0.000, C 0.000 }
gfCNCPoint2[7073] = {X 572.3399, Y 61.1017, Z -3.0000, A 0.000, B 0.000, C 0.000 }
gfCNCPoint2[7074] = {X 570.7903, Y 61.3253, Z -3.0000, A 0.000, B 0.000, C 0.000 }
gfCNCPoint2[7075] = {X 569.2264, Y 61.4000, Z -3.0000, A 0.000, B 0.000, C 0.000 }
gfCNCPoint2[7076] = {X 562.4443, Y 61.4000, Z -3.0000, A 0.000, B 0.000, C 0.000 }
gfCNCPoint2[7077] = {X 560.5828, Y 61.2940, Z -3.0000, A 0.000, B 0.000, C 0.000 }
gfCNCPoint2[7078] = {X 558.7453, Y 60.9774, Z -3.0000, A 0.000, B 0.000, C 0.000 }
gfCNCPoint2[7079] = {X 556.9557, Y 60.4543, Z -3.0000, A 0.000, B 0.000, C 0.000 }
gfCNCPoint2[7080] = {X 555.2370, Y 59.7314, Z -3.0000, A 0.000, B 0.000, C 0.000 }
gfCNCPoint2[7081] = {X 553.6114, Y 58.8181, Z -3.0000, A 0.000, B 0.000, C 0.000 }
gfCNCPoint2[7082] = {X 552.1001, Y 57.7262, Z -3.0000, A 0.000, B 0.000, C 0.000 }
gfCNCPoint2[7083] = {X 550.7224, Y 56.4698, Z -3.0000, A 0.000, B 0.000, C 0.000 }
gfCNCPoint2[7084] = {X 549.4963, Y 55.0652, Z -3.0000, A 0.000, B 0.000, C 0.000 }
gfCNCPoint2[7085] = {X 548.4375, Y 53.5304, Z -3.0000, A 0.000, B 0.000, C 0.000 }
gfCNCPoint2[7086] = {X 547.3157, Y 54.0419, Z -3.0000, A 0.000, B 0.000, C 0.000 }
gfCNCPoint2[7087] = {X 546.1380, Y 54.4068, Z -3.0000, A 0.000, B 0.000, C 0.000 }
gfCNCPoint2[7088] = {X 544.9236, Y 54.6190, Z -3.0000, A 0.000, B 0.000, C 0.000 }
gfCNCPoint2[7089] = {X 543.6920, Y 54.6753, Z -3.0000, A 0.000, B 0.000, C 0.000 }
gfCNCPoint2[7090] = {X 526.1843, Y 54.6757, Z -3.0000, A 0.000, B 0.000, C 0.000 }
gfCNCPoint2[7091] = {X 524.8903, Y 55.4724, Z -3.0000, A 0.000, B 0.000, C 0.000 }
gfCNCPoint2[7092] = {X 523.4890, Y 56.0603, Z -3.0000, A 0.000, B 0.000, C 0.000 }
gfCNCPoint2[7093] = {X 522.0140, Y 56.4255, Z -3.0000, A 0.000, B 0.000, C 0.000 }
gfCNCPoint2[7094] = {X 520.5003, Y 56.5591, Z -3.0000, A 0.000, B 0.000, C 0.000 }
gfCNCPoint2[7095] = {X 519.7998, Y 56.5591, Z -3.0000, A 0.000, B 0.000, C 0.000 }
gfCNCPoint2[7096] = {X 518.3493, Y 56.4498, Z -3.0000, A 0.000, B 0.000, C 0.000 }
gfCNCPoint2[7097] = {X 516.9316, Y 56.1244, Z -3.0000, A 0.000, B 0.000, C 0.000 }
gfCNCPoint2[7098] = {X 515.5787, Y 55.5903, Z -3.0000, A 0.000, B 0.000, C 0.000 }
gfCNCPoint2[7099] = {X 514.3210, Y 54.8595, Z -3.0000, A 0.000, B 0.000, C 0.000 }
gfCNCPoint2[7100] = {X 513.1871, Y 53.9484, Z -3.0000, A 0.000, B 0.000, C 0.000 }
gfCNCPoint2[7101] = {X 512.2025, Y 52.8778, Z -3.0000, A 0.000, B 0.000, C 0.000 }
gfCNCPoint2[7102] = {X 511.3855, Y 51.6648, Z -3.0000, A 0.000, B 0.000, C 0.000 }
gfCNCPoint2[7103] = {X 510.7606, Y 50.3426, Z -3.0000, A 0.000, B 0.000, C 0.000 }
gfCNCPoint2[7104] = {X 509.8636, Y 51.4977, Z -3.0000, A 0.000, B 0.000, C 0.000 }
gfCNCPoint2[7105] = {X 508.8029, Y 52.5044, Z -3.0000, A 0.000, B 0.000, C 0.000 }
gfCNCPoint2[7106] = {X 507.7229, Y 53.2678, Z -3.0000, A 0.000, B 0.000, C 0.000 }
gfCNCPoint2[7107] = {X 506.5489, Y 53.8769, Z -3.0000, A 0.000, B 0.000, C 0.000 }
gfCNCPoint2[7108] = {X 505.3028, Y 54.3203, Z -3.0000, A 0.000, B 0.000, C 0.000 }
gfCNCPoint2[7109] = {X 504.0080, Y 54.5896, Z -3.0000, A 0.000, B 0.000, C 0.000 }
gfCNCPoint2[7110] = {X 502.6885, Y 54.6800, Z -3.0000, A 0.000, B 0.000, C 0.000 }
gfCNCPoint2[7111] = {X 496.2450, Y 54.6800, Z -3.0000, A 0.000, B 0.000, C 0.000 }
gfCNCPoint2[7112] = {X 495.0285, Y 54.6033, Z -3.0000, A 0.000, B 0.000, C 0.000 }
gfCNCPoint2[7113] = {X 493.8313, Y 54.3742, Z -3.0000, A 0.000, B 0.000, C 0.000 }
gfCNCPoint2[7114] = {X 492.6724, Y 53.9966, Z -3.0000, A 0.000, B 0.000, C 0.000 }
gfCNCPoint2[7115] = {X 491.4451, Y 53.4062, Z -3.0000, A 0.000, B 0.000, C 0.000 }
gfCNCPoint2[7116] = {X 490.3129, Y 52.6493, Z -3.0000, A 0.000, B 0.000, C 0.000 }
gfCNCPoint2[7117] = {X 489.2980, Y 51.7410, Z -3.0000, A 0.000, B 0.000, C 0.000 }
gfCNCPoint2[7118] = {X 488.8683, Y 52.1573, Z -3.0000, A 0.000, B 0.000, C 0.000 }
gfCNCPoint2[7119] = {X 488.4137, Y 52.5463, Z -3.0000, A 0.000, B 0.000, C 0.000 }
gfCNCPoint2[7120] = {X 488.8649, Y 53.8245, Z -3.0000, A 0.000, B 0.000, C 0.000 }
gfCNCPoint2[7121] = {X 489.1946, Y 55.1393, Z -3.0000, A 0.000, B 0.000, C 0.000 }
gfCNCPoint2[7122] = {X 489.3999, Y 56.4792, Z -3.0000, A 0.000, B 0.000, C 0.000 }
gfCNCPoint2[7123] = {X 489.4600, Y 57.2386, Z -3.0000, A 0.000, B 0.000, C 0.000 }
gfCNCPoint2[7124] = {X 489.4800, Y 58.0000, Z -3.0000, A 0.000, B 0.000, C 0.000 }
gfCNCPoint2[7125] = {X 489.4795, Y 59.0537, Z -3.0000, A 0.000, B 0.000, C 0.000 }
gfCNCPoint2[7126] = {X 489.3595, Y 60.7979, Z -3.0000, A 0.000, B 0.000, C 0.000 }
gfCNCPoint2[7127] = {X 489.0303, Y 62.5149, Z -3.0000, A 0.000, B 0.000, C 0.000 }
gfCNCPoint2[7128] = {X 488.4964, Y 64.1797, Z -3.0000, A 0.000, B 0.000, C 0.000 }
gfCNCPoint2[7129] = {X 487.7659, Y 65.7680, Z -3.0000, A 0.000, B 0.000, C 0.000 }
gfCNCPoint2[7130] = {X 486.8492, Y 67.2567, Z -3.0000, A 0.000, B 0.000, C 0.000 }
gfCNCPoint2[7131] = {X 485.7598, Y 68.6241, Z -3.0000, A 0.000, B 0.000, C 0.000 }
gfCNCPoint2[7132] = {X 485.7601, Y 87.3799, Z -3.0000, A 0.000, B 0.000, C 0.000 }
gfCNCPoint2[7133] = {X 486.0679, Y 87.7325, Z -3.0000, A 0.000, B 0.000, C 0.000 }
gfCNCPoint2[7134] = {X 486.3641, Y 88.0950, Z -3.0000, A 0.000, B 0.000, C 0.000 }
gfCNCPoint2[7135] = {X 507.6818, Y 88.0950, Z -3.0000, A 0.000, B 0.000, C 0.000 }
gfCNCPoint2[7136] = {X 507.6818, Y 90.4950, Z -3.0000, A 0.000, B 0.000, C 0.000 }
gfCNCPoint2[7137] = {X 590.4965, Y 90.4950, Z -3.0000, A 0.000, B 0.000, C 0.000 }
gfCNCPoint2[7138] = {X 590.4965, Y 58.6615, Z -3.0000, A 0.000, B 0.000, C 0.000 }
gfCNCPoint2[7139] = {X 588.9715, Y 58.2279, Z -3.0000, A 0.000, B 0.000, C 0.000 }
gfCNCPoint2[7140] = {X 587.5052, Y 57.6246, Z -3.0000, A 0.000, B 0.000, C 0.000 }
gfCNCPoint2[7141] = {X 585.8387, Y 58.2956, Z -3.0000, A 0.000, B 0.000, C 0.000 }
gfCNCPoint2[7142] = {X 584.0999, Y 58.7477, Z -3.0000, A 0.000, B 0.000, C 0.000 }
gfCNCPoint2[7143] = {X 582.3176, Y 58.9733, Z -3.0000, A 0.000, B 0.000, C 0.000 }
gfCNCPoint2[7144] = {X 580.5210, Y 58.9689, Z -3.0000, A 0.000, B 0.000, C 0.000 }
gfCNCPoint2[7145] = {X 578.7398, Y 58.7344, Z -3.0000, A 0.000, B 0.000, C 0.000 }
gfCNCPoint2[7146] = {X 577.0034, Y 58.2738, Z -3.0000, A 0.000, B 0.000, C 0.000 }
gfCNCPoint2[7147] = {X 575.3401, Y 57.5945, Z -3.0000, A 0.000, B 0.000, C 0.000 }
gfCNCPoint2[7148] = {X 573.8813, Y 58.2035, Z -3.0000, A 0.000, B 0.000, C 0.000 }
gfCNCPoint2[7149] = {X 572.3630, Y 58.6441, Z -3.0000, A 0.000, B 0.000, C 0.000 }
gfCNCPoint2[7150] = {X 570.8048, Y 58.9107, Z -3.0000, A 0.000, B 0.000, C 0.000 }
gfCNCPoint2[7151] = {X 569.2264, Y 59.0000, Z -3.0000, A 0.000, B 0.000, C 0.000 }
gfCNCPoint2[7152] = {X 562.4443, Y 59.0000, Z -3.0000, A 0.000, B 0.000, C 0.000 }
gfCNCPoint2[7153] = {X 560.6576, Y 58.8855, Z -3.0000, A 0.000, B 0.000, C 0.000 }
gfCNCPoint2[7154] = {X 558.9001, Y 58.5439, Z -3.0000, A 0.000, B 0.000, C 0.000 }
gfCNCPoint2[7155] = {X 557.2006, Y 57.9809, Z -3.0000, A 0.000, B 0.000, C 0.000 }
gfCNCPoint2[7156] = {X 555.5868, Y 57.2055, Z -3.0000, A 0.000, B 0.000, C 0.000 }
gfCNCPoint2[7157] = {X 554.0852, Y 56.2305, Z -3.0000, A 0.000, B 0.000, C 0.000 }
gfCNCPoint2[7158] = {X 552.7203, Y 55.0719, Z -3.0000, A 0.000, B 0.000, C 0.000 }
gfCNCPoint2[7159] = {X 551.5144, Y 53.7485, Z -3.0000, A 0.000, B 0.000, C 0.000 }
gfCNCPoint2[7160] = {X 550.4872, Y 52.2821, Z -3.0000, A 0.000, B 0.000, C 0.000 }
gfCNCPoint2[7161] = {X 549.8375, Y 51.0884, Z -3.0000, A 0.000, B 0.000, C 0.000 }
gfCNCPoint2[7162] = {X 549.3066, Y 49.8373, Z -3.0000, A 0.000, B 0.000, C 0.000 }
gfCNCPoint2[7163] = {X 548.3752, Y 50.7142, Z -3.0000, A 0.000, B 0.000, C 0.000 }
gfCNCPoint2[7164] = {X 547.3048, Y 51.4145, Z -3.0000, A 0.000, B 0.000, C 0.000 }
gfCNCPoint2[7165] = {X 546.1633, Y 51.9054, Z -3.0000, A 0.000, B 0.000, C 0.000 }
gfCNCPoint2[7166] = {X 544.9551, Y 52.1951, Z -3.0000, A 0.000, B 0.000, C 0.000 }
gfCNCPoint2[7167] = {X 543.7151, Y 52.2753, Z -3.0000, A 0.000, B 0.000, C 0.000 }
gfCNCPoint2[7168] = {X 525.3420, Y 52.2757, Z -3.0000, A 0.000, B 0.000, C 0.000 }
gfCNCPoint2[7169] = {X 524.2750, Y 53.0673, Z -3.0000, A 0.000, B 0.000, C 0.000 }
gfCNCPoint2[7170] = {X 523.0841, Y 53.6564, Z -3.0000, A 0.000, B 0.000, C 0.000 }
gfCNCPoint2[7171] = {X 521.8074, Y 54.0243, Z -3.0000, A 0.000, B 0.000, C 0.000 }
gfCNCPoint2[7172] = {X 520.4856, Y 54.1591, Z -3.0000, A 0.000, B 0.000, C 0.000 }
gfCNCPoint2[7173] = {X 519.7998, Y 54.1591, Z -3.0000, A 0.000, B 0.000, C 0.000 }
gfCNCPoint2[7174] = {X 518.5529, Y 54.0515, Z -3.0000, A 0.000, B 0.000, C 0.000 }
gfCNCPoint2[7175] = {X 517.3428, Y 53.7320, Z -3.0000, A 0.000, B 0.000, C 0.000 }
gfCNCPoint2[7176] = {X 516.2054, Y 53.2099, Z -3.0000, A 0.000, B 0.000, C 0.000 }
gfCNCPoint2[7177] = {X 515.1742, Y 52.5007, Z -3.0000, A 0.000, B 0.000, C 0.000 }
gfCNCPoint2[7178] = {X 514.2797, Y 51.6254, Z -3.0000, A 0.000, B 0.000, C 0.000 }
gfCNCPoint2[7179] = {X 513.5483, Y 50.6098, Z -3.0000, A 0.000, B 0.000, C 0.000 }
gfCNCPoint2[7180] = {X 513.0017, Y 49.4839, Z -3.0000, A 0.000, B 0.000, C 0.000 }
gfCNCPoint2[7181] = {X 512.7353, Y 48.6374, Z -3.0000, A 0.000, B 0.000, C 0.000 }
gfCNCPoint2[7182] = {X 512.5739, Y 47.7649, Z -3.0000, A 0.000, B 0.000, C 0.000 }
gfCNCPoint2[7183] = {X 512.5198, Y 46.8791, Z -3.0000, A 0.000, B 0.000, C 0.000 }
gfCNCPoint2[7184] = {X 512.5198, Y 39.9011, Z -3.0000, A 0.000, B 0.000, C 0.000 }
gfCNCPoint2[7185] = {X 512.5807, Y 38.9614, Z -3.0000, A 0.000, B 0.000, C 0.000 }
gfCNCPoint2[7186] = {X 512.7624, Y 38.0374, Z -3.0000, A 0.000, B 0.000, C 0.000 }
gfCNCPoint2[7187] = {X 513.0618, Y 37.1446, Z -3.0000, A 0.000, B 0.000, C 0.000 }
gfCNCPoint2[7188] = {X 513.5574, Y 36.1554, Z -3.0000, A 0.000, B 0.000, C 0.000 }
gfCNCPoint2[7189] = {X 514.1970, Y 35.2527, Z -3.0000, A 0.000, B 0.000, C 0.000 }
gfCNCPoint2[7190] = {X 514.9661, Y 34.4574, Z -3.0000, A 0.000, B 0.000, C 0.000 }
gfCNCPoint2[7191] = {X 515.8469, Y 33.7878, Z -3.0000, A 0.000, B 0.000, C 0.000 }
gfCNCPoint2[7192] = {X 513.2406, Y 29.7570, Z -3.0000, A 0.000, B 0.000, C 0.000 }
gfCNCPoint2[7193] = {X 513.5213, Y 29.5809, Z -3.0000, A 0.000, B 0.000, C 0.000 }
gfCNCPoint2[7194] = {X 513.8068, Y 29.4125, Z -3.0000, A 0.000, B 0.000, C 0.000 }
gfCNCPoint2[7195] = {X 513.8068, Y 27.6757, Z -3.0000, A 0.000, B 0.000, C 0.000 }
gfCNCPoint2[7196] = {X 513.5212, Y 27.5009, Z -3.0000, A 0.000, B 0.000, C 0.000 }
gfCNCPoint2[7197] = {X 513.2406, Y 27.3183, Z -3.0000, A 0.000, B 0.000, C 0.000 }
gfCNCPoint2[7198] = {X 513.2406, Y 29.7570, Z -3.0000, A 0.000, B 0.000, C 0.000 }
gfCNCPoint2[7199] = {X 514.5437, Y 31.7724, Z -3.0000, A 0.000, B 0.000, C 0.000 }
gfCNCPoint2[7200] = {X 515.3544, Y 31.3022, Z -3.0000, A 0.000, B 0.000, C 0.000 }
gfCNCPoint2[7201] = {X 516.2068, Y 30.9126, Z -3.0000, A 0.000, B 0.000, C 0.000 }
gfCNCPoint2[7202] = {X 516.2068, Y 26.2046, Z -3.0000, A 0.000, B 0.000, C 0.000 }
gfCNCPoint2[7203] = {X 515.3710, Y 25.8039, Z -3.0000, A 0.000, B 0.000, C 0.000 }
gfCNCPoint2[7204] = {X 514.5774, Y 25.3251, Z -3.0000, A 0.000, B 0.000, C 0.000 }
gfCNCPoint2[7205] = {X 513.5940, Y 24.5700, Z -3.0000, A 0.000, B 0.000, C 0.000 }
gfCNCPoint2[7206] = {X 512.7152, Y 23.6953, Z -3.0000, A 0.000, B 0.000, C 0.000 }
gfCNCPoint2[7207] = {X 511.9554, Y 22.7156, Z -3.0000, A 0.000, B 0.000, C 0.000 }
gfCNCPoint2[7208] = {X 511.3271, Y 21.6467, Z -3.0000, A 0.000, B 0.000, C 0.000 }
gfCNCPoint2[7209] = {X 510.8406, Y 20.5063, Z -3.0000, A 0.000, B 0.000, C 0.000 }
gfCNCPoint2[7210] = {X 510.8405, Y 36.2358, Z -3.0000, A 0.000, B 0.000, C 0.000 }
gfCNCPoint2[7211] = {X 511.4994, Y 34.9205, Z -3.0000, A 0.000, B 0.000, C 0.000 }
gfCNCPoint2[7212] = {X 512.3500, Y 33.7202, Z -3.0000, A 0.000, B 0.000, C 0.000 }
gfCNCPoint2[7213] = {X 513.3726, Y 32.6627, Z -3.0000, A 0.000, B 0.000, C 0.000 }
gfCNCPoint2[7214] = {X 514.5437, Y 31.7724, Z -3.0000, A 0.000, B 0.000, C 0.000 }
gfCNCPoint2[7215] = {X 515.8469, Y 33.7878, Z -3.0000, A 0.000, B 0.000, C 0.000 }
gfCNCPoint2[7216] = {X 516.7435, Y 33.2937, Z -3.0000, A 0.000, B 0.000, C 0.000 }
gfCNCPoint2[7217] = {X 517.7005, Y 32.9303, Z -3.0000, A 0.000, B 0.000, C 0.000 }
gfCNCPoint2[7218] = {X 518.6990, Y 32.7048, Z -3.0000, A 0.000, B 0.000, C 0.000 }
gfCNCPoint2[7219] = {X 518.6299, Y 32.1290, Z -3.0000, A 0.000, B 0.000, C 0.000 }
gfCNCPoint2[7220] = {X 518.6068, Y 31.5495, Z -3.0000, A 0.000, B 0.000, C 0.000 }
gfCNCPoint2[7221] = {X 518.6068, Y 24.5714, Z -3.0000, A 0.000, B 0.000, C 0.000 }
gfCNCPoint2[7222] = {X 518.6080, Y 24.4373, Z -3.0000, A 0.000, B 0.000, C 0.000 }
gfCNCPoint2[7223] = {X 517.3909, Y 24.0939, Z -3.0000, A 0.000, B 0.000, C 0.000 }
gfCNCPoint2[7224] = {X 516.2517, Y 23.5450, Z -3.0000, A 0.000, B 0.000, C 0.000 }
gfCNCPoint2[7225] = {X 515.2246, Y 22.8073, Z -3.0000, A 0.000, B 0.000, C 0.000 }
gfCNCPoint2[7226] = {X 514.3407, Y 21.9030, Z -3.0000, A 0.000, B 0.000, C 0.000 }
gfCNCPoint2[7227] = {X 513.6266, Y 20.8593, Z -3.0000, A 0.000, B 0.000, C 0.000 }
gfCNCPoint2[7228] = {X 513.1038, Y 19.7078, Z -3.0000, A 0.000, B 0.000, C 0.000 }
gfCNCPoint2[7229] = {X 512.7935, Y 18.5144, Z -3.0000, A 0.000, B 0.000, C 0.000 }
gfCNCPoint2[7230] = {X 512.6891, Y 17.2857, Z -3.0000, A 0.000, B 0.000, C 0.000 }
gfCNCPoint2[7231] = {X 512.6891, Y 10.3077, Z -3.0000, A 0.000, B 0.000, C 0.000 }
gfCNCPoint2[7232] = {X 512.7002, Y 9.9058, Z -3.0000, A 0.000, B 0.000, C 0.000 }
gfCNCPoint2[7233] = {X 512.7335, Y 9.5050, Z -3.0000, A 0.000, B 0.000, C 0.000 }
gfCNCPoint2[7234] = {X 509.4581, Y 9.5050, Z -3.0000, A 0.000, B 0.000, C 0.000 }
gfCNCPoint2[7235] = {X 509.7401, Y 10.3729, Z -3.0000, A 0.000, B 0.000, C 0.000 }
gfCNCPoint2[7236] = {X 509.9112, Y 11.2692, Z -3.0000, A 0.000, B 0.000, C 0.000 }
gfCNCPoint2[7237] = {X 509.9685, Y 12.1800, Z -3.0000, A 0.000, B 0.000, C 0.000 }
gfCNCPoint2[7238] = {X 509.9682, Y 13.0462, Z -3.0000, A 0.000, B 0.000, C 0.000 }
gfCNCPoint2[7239] = {X 509.8611, Y 14.2238, Z -3.0000, A 0.000, B 0.000, C 0.000 }
gfCNCPoint2[7240] = {X 509.5648, Y 15.3685, Z -3.0000, A 0.000, B 0.000, C 0.000 }
gfCNCPoint2[7241] = {X 509.0871, Y 16.4502, Z -3.0000, A 0.000, B 0.000, C 0.000 }
gfCNCPoint2[7242] = {X 508.4406, Y 17.4403, Z -3.0000, A 0.000, B 0.000, C 0.000 }
gfCNCPoint2[7243] = {X 508.4405, Y 39.7465, Z -3.0000, A 0.000, B 0.000, C 0.000 }
gfCNCPoint2[7244] = {X 509.0889, Y 40.7399, Z -3.0000, A 0.000, B 0.000, C 0.000 }
gfCNCPoint2[7245] = {X 509.5673, Y 41.8254, Z -3.0000, A 0.000, B 0.000, C 0.000 }
gfCNCPoint2[7246] = {X 509.8630, Y 42.9742, Z -3.0000, A 0.000, B 0.000, C 0.000 }
gfCNCPoint2[7247] = {X 509.9683, Y 44.1558, Z -3.0000, A 0.000, B 0.000, C 0.000 }
gfCNCPoint2[7248] = {X 509.9685, Y 45.0000, Z -3.0000, A 0.000, B 0.000, C 0.000 }
